gfCNCPoint2[8454] = {X 428.4411, Y 41.5212, Z -3.0000, A 0.000, B 0.000, C 0.000 }
gfCNCPoint2[8455] = {X 429.0371, Y 40.7849, Z -3.0000, A 0.000, B 0.000, C 0.000 }
gfCNCPoint2[8456] = {X 429.7641, Y 40.1776, Z -3.0000, A 0.000, B 0.000, C 0.000 }
gfCNCPoint2[8457] = {X 430.5947, Y 39.7222, Z -3.0000, A 0.000, B 0.000, C 0.000 }
gfCNCPoint2[8458] = {X 434.2534, Y 32.5608, Z -3.0000, A 0.000, B 0.000, C 0.000 }
gfCNCPoint2[8459] = {X 432.9191, Y 31.5580, Z -3.0000, A 0.000, B 0.000, C 0.000 }
gfCNCPoint2[8460] = {X 431.7385, Y 30.3782, Z -3.0000, A 0.000, B 0.000, C 0.000 }
gfCNCPoint2[8461] = {X 430.7348, Y 29.0445, Z -3.0000, A 0.000, B 0.000, C 0.000 }
gfCNCPoint2[8462] = {X 429.9280, Y 27.5834, Z -3.0000, A 0.000, B 0.000, C 0.000 }
gfCNCPoint2[8463] = {X 429.3339, Y 26.0236, Z -3.0000, A 0.000, B 0.000, C 0.000 }
gfCNCPoint2[8464] = {X 428.8998, Y 24.1501, Z -3.0000, A 0.000, B 0.000, C 0.000 }
gfCNCPoint2[8465] = {X 428.6784, Y 22.2397, Z -3.0000, A 0.000, B 0.000, C 0.000 }
gfCNCPoint2[8466] = {X 428.6725, Y 20.3166, Z -3.0000, A 0.000, B 0.000, C 0.000 }
gfCNCPoint2[8467] = {X 428.8821, Y 18.4049, Z -3.0000, A 0.000, B 0.000, C 0.000 }
gfCNCPoint2[8468] = {X 429.3046, Y 16.5287, Z -3.0000, A 0.000, B 0.000, C 0.000 }
gfCNCPoint2[8469] = {X 429.8216, Y 15.0577, Z -3.0000, A 0.000, B 0.000, C 0.000 }
gfCNCPoint2[8470] = {X 430.5198, Y 13.6635, Z -3.0000, A 0.000, B 0.000, C 0.000 }
gfCNCPoint2[8471] = {X 431.3881, Y 12.3684, Z -3.0000, A 0.000, B 0.000, C 0.000 }
gfCNCPoint2[8472] = {X 432.4125, Y 11.1930, Z -3.0000, A 0.000, B 0.000, C 0.000 }
gfCNCPoint2[8473] = {X 433.6947, Y 10.0649, Z -3.0000, A 0.000, B 0.000, C 0.000 }
gfCNCPoint2[8474] = {X 435.1201, Y 9.1243, Z -3.0000, A 0.000, B 0.000, C 0.000 }
gfCNCPoint2[8475] = {X 436.6617, Y 8.3894, Z -3.0000, A 0.000, B 0.000, C 0.000 }
gfCNCPoint2[8476] = {X 438.2899, Y 7.8741, Z -3.0000, A 0.000, B 0.000, C 0.000 }
gfCNCPoint2[8477] = {X 439.9586, Y 7.5566, Z -3.0000, A 0.000, B 0.000, C 0.000 }
gfCNCPoint2[8478] = {X 441.6469, Y 7.3699, Z -3.0000, A 0.000, B 0.000, C 0.000 }
gfCNCPoint2[8479] = {X 443.3446, Y 7.3153, Z -3.0000, A 0.000, B 0.000, C 0.000 }
gfCNCPoint2[8480] = {X 459.4466, Y 7.3112, Z -3.0000, A 0.000, B 0.000, C 0.000 }
gfCNCPoint2[8481] = {X 460.4094, Y 7.4073, Z -3.0000, A 0.000, B 0.000, C 0.000 }
gfCNCPoint2[8482] = {X 461.3341, Y 7.6918, Z -3.0000, A 0.000, B 0.000, C 0.000 }
gfCNCPoint2[8483] = {X 462.1845, Y 8.1534, Z -3.0000, A 0.000, B 0.000, C 0.000 }
gfCNCPoint2[8484] = {X 462.9268, Y 8.7740, Z -3.0000, A 0.000, B 0.000, C 0.000 }
gfCNCPoint2[8485] = {X 463.5318, Y 9.5291, Z -3.0000, A 0.000, B 0.000, C 0.000 }
gfCNCPoint2[8486] = {X 463.9756, Y 10.3888, Z -3.0000, A 0.000, B 0.000, C 0.000 }
gfCNCPoint2[8487] = {X 464.2316, Y 11.2695, Z -3.0000, A 0.000, B 0.000, C 0.000 }
gfCNCPoint2[8488] = {X 464.3179, Y 12.1826, Z -3.0000, A 0.000, B 0.000, C 0.000 }
gfCNCPoint2[8489] = {X 464.3179, Y 12.9779, Z -3.0000, A 0.000, B 0.000, C 0.000 }
gfCNCPoint2[8490] = {X 464.2173, Y 13.9638, Z -3.0000, A 0.000, B 0.000, C 0.000 }
gfCNCPoint2[8491] = {X 463.9196, Y 14.9091, Z -3.0000, A 0.000, B 0.000, C 0.000 }
gfCNCPoint2[8492] = {X 463.4371, Y 15.7747, Z -3.0000, A 0.000, B 0.000, C 0.000 }
gfCNCPoint2[8493] = {X 462.7896, Y 16.5249, Z -3.0000, A 0.000, B 0.000, C 0.000 }
gfCNCPoint2[8494] = {X 462.7893, Y 16.7698, Z -3.0000, A 0.000, B 0.000, C 0.000 }
gfCNCPoint2[8495] = {X 462.7904, Y 40.6626, Z -3.0000, A 0.000, B 0.000, C 0.000 }
gfCNCPoint2[8496] = {X 463.4315, Y 41.4042, Z -3.0000, A 0.000, B 0.000, C 0.000 }
gfCNCPoint2[8497] = {X 463.9115, Y 42.2590, Z -3.0000, A 0.000, B 0.000, C 0.000 }
gfCNCPoint2[8498] = {X 464.2109, Y 43.1925, Z -3.0000, A 0.000, B 0.000, C 0.000 }
gfCNCPoint2[8499] = {X 464.3178, Y 44.1670, Z -3.0000, A 0.000, B 0.000, C 0.000 }
gfCNCPoint2[8500] = {X 464.3179, Y 45.0000, Z -3.0000, A 0.000, B 0.000, C 0.000 }
gfCNCPoint2[8501] = {X 464.3082, Y 45.3090, Z -3.0000, A 0.000, B 0.000, C 0.000 }
gfCNCPoint2[8502] = {X 464.2788, Y 45.6167, Z -3.0000, A 0.000, B 0.000, C 0.000 }
gfCNCPoint2[8503] = {X 464.0485, Y 46.5992, Z -3.0000, A 0.000, B 0.000, C 0.000 }
gfCNCPoint2[8504] = {X 463.6209, Y 47.5134, Z -3.0000, A 0.000, B 0.000, C 0.000 }
gfCNCPoint2[8505] = {X 463.0145, Y 48.3200, Z -3.0000, A 0.000, B 0.000, C 0.000 }
gfCNCPoint2[8506] = {X 462.6627, Y 47.9934, Z -3.0000, A 0.000, B 0.000, C 0.000 }
gfCNCPoint2[8507] = {X 461.9835, Y 48.5889, Z -3.0000, A 0.000, B 0.000, C 0.000 }
gfCNCPoint2[8508] = {X 461.1970, Y 49.0331, Z -3.0000, A 0.000, B 0.000, C 0.000 }
gfCNCPoint2[8509] = {X 460.3364, Y 49.3073, Z -3.0000, A 0.000, B 0.000, C 0.000 }
gfCNCPoint2[8510] = {X 459.4379, Y 49.4000, Z -3.0000, A 0.000, B 0.000, C 0.000 }
gfCNCPoint2[8511] = {X 452.9945, Y 49.4000, Z -3.0000, A 0.000, B 0.000, C 0.000 }
gfCNCPoint2[8512] = {X 452.0154, Y 49.2897, Z -3.0000, A 0.000, B 0.000, C 0.000 }
gfCNCPoint2[8513] = {X 451.0854, Y 48.9643, Z -3.0000, A 0.000, B 0.000, C 0.000 }
gfCNCPoint2[8514] = {X 450.2511, Y 48.4400, Z -3.0000, A 0.000, B 0.000, C 0.000 }
gfCNCPoint2[8515] = {X 449.5544, Y 47.7433, Z -3.0000, A 0.000, B 0.000, C 0.000 }
gfCNCPoint2[8516] = {X 449.0302, Y 46.9091, Z -3.0000, A 0.000, B 0.000, C 0.000 }
gfCNCPoint2[8517] = {X 448.7048, Y 45.9791, Z -3.0000, A 0.000, B 0.000, C 0.000 }
gfCNCPoint2[8518] = {X 448.5945, Y 45.0000, Z -3.0000, A 0.000, B 0.000, C 0.000 }
gfCNCPoint2[8519] = {X 448.5949, Y 44.1483, Z -3.0000, A 0.000, B 0.000, C 0.000 }
gfCNCPoint2[8520] = {X 448.7053, Y 43.2275, Z -3.0000, A 0.000, B 0.000, C 0.000 }
gfCNCPoint2[8521] = {X 449.0063, Y 42.3503, Z -3.0000, A 0.000, B 0.000, C 0.000 }
gfCNCPoint2[8522] = {X 449.4844, Y 41.5556, Z -3.0000, A 0.000, B 0.000, C 0.000 }
gfCNCPoint2[8523] = {X 450.1184, Y 40.8789, Z -3.0000, A 0.000, B 0.000, C 0.000 }
gfCNCPoint2[8524] = {X 450.1184, Y 34.5538, Z -3.0000, A 0.000, B 0.000, C 0.000 }
gfCNCPoint2[8525] = {X 447.5228, Y 34.5538, Z -3.0000, A 0.000, B 0.000, C 0.000 }
gfCNCPoint2[8526] = {X 443.2762, Y 42.8220, Z -3.0000, A 0.000, B 0.000, C 0.000 }
gfCNCPoint2[8527] = {X 443.4440, Y 43.5064, Z -3.0000, A 0.000, B 0.000, C 0.000 }
gfCNCPoint2[8528] = {X 443.5005, Y 44.2089, Z -3.0000, A 0.000, B 0.000, C 0.000 }
gfCNCPoint2[8529] = {X 443.5005, Y 45.0000, Z -3.0000, A 0.000, B 0.000, C 0.000 }
gfCNCPoint2[8530] = {X 443.3902, Y 45.9791, Z -3.0000, A 0.000, B 0.000, C 0.000 }
gfCNCPoint2[8531] = {X 443.0647, Y 46.9091, Z -3.0000, A 0.000, B 0.000, C 0.000 }
gfCNCPoint2[8532] = {X 442.5405, Y 47.7434, Z -3.0000, A 0.000, B 0.000, C 0.000 }
gfCNCPoint2[8533] = {X 441.8438, Y 48.4401, Z -3.0000, A 0.000, B 0.000, C 0.000 }
gfCNCPoint2[8534] = {X 441.0096, Y 48.9643, Z -3.0000, A 0.000, B 0.000, C 0.000 }
gfCNCPoint2[8535] = {X 440.0796, Y 49.2897, Z -3.0000, A 0.000, B 0.000, C 0.000 }
gfCNCPoint2[8536] = {X 439.1005, Y 49.4000, Z -3.0000, A 0.000, B 0.000, C 0.000 }
gfCNCPoint2[8537] = {X 432.5144, Y 49.4000, Z -3.0000, A 0.000, B 0.000, C 0.000 }
gfCNCPoint2[8538] = {X 431.5353, Y 49.2897, Z -3.0000, A 0.000, B 0.000, C 0.000 }
gfCNCPoint2[8539] = {X 430.6053, Y 48.9643, Z -3.0000, A 0.000, B 0.000, C 0.000 }
gfCNCPoint2[8540] = {X 429.7711, Y 48.4401, Z -3.0000, A 0.000, B 0.000, C 0.000 }
gfCNCPoint2[8541] = {X 429.0743, Y 47.7434, Z -3.0000, A 0.000, B 0.000, C 0.000 }
gfCNCPoint2[8542] = {X 428.5501, Y 46.9091, Z -3.0000, A 0.000, B 0.000, C 0.000 }
gfCNCPoint2[8543] = {X 428.2247, Y 45.9791, Z -3.0000, A 0.000, B 0.000, C 0.000 }
gfCNCPoint2[8544] = {X 428.1144, Y 45.0000, Z -3.0000, A 0.000, B 0.000, C 0.000 }
gfCNCPoint2[8545] = {X 428.1148, Y 44.1483, Z -3.0000, A 0.000, B 0.000, C 0.000 }
gfCNCPoint2[8546] = {X 428.2132, Y 43.2816, Z -3.0000, A 0.000, B 0.000, C 0.000 }
gfCNCPoint2[8547] = {X 428.4806, Y 42.4514, Z -3.0000, A 0.000, B 0.000, C 0.000 }
gfCNCPoint2[8548] = {X 428.9065, Y 41.6903, Z -3.0000, A 0.000, B 0.000, C 0.000 }
gfCNCPoint2[8549] = {X 429.4741, Y 41.0281, Z -3.0000, A 0.000, B 0.000, C 0.000 }
gfCNCPoint2[8550] = {X 430.1613, Y 40.4909, Z -3.0000, A 0.000, B 0.000, C 0.000 }
gfCNCPoint2[8551] = {X 430.9408, Y 40.0998, Z -3.0000, A 0.000, B 0.000, C 0.000 }
gfCNCPoint2[8552] = {X 434.8818, Y 32.3858, Z -3.0000, A 0.000, B 0.000, C 0.000 }
gfCNCPoint2[8553] = {X 433.7183, Y 31.5933, Z -3.0000, A 0.000, B 0.000, C 0.000 }
gfCNCPoint2[8554] = {X 432.6614, Y 30.6634, Z -3.0000, A 0.000, B 0.000, C 0.000 }
gfCNCPoint2[8555] = {X 431.7272, Y 29.6103, Z -3.0000, A 0.000, B 0.000, C 0.000 }
gfCNCPoint2[8556] = {X 430.9298, Y 28.4502, Z -3.0000, A 0.000, B 0.000, C 0.000 }
gfCNCPoint2[8557] = {X 430.2815, Y 27.2006, Z -3.0000, A 0.000, B 0.000, C 0.000 }
gfCNCPoint2[8558] = {X 429.7922, Y 25.8807, Z -3.0000, A 0.000, B 0.000, C 0.000 }
gfCNCPoint2[8559] = {X 429.3715, Y 24.0610, Z -3.0000, A 0.000, B 0.000, C 0.000 }
gfCNCPoint2[8560] = {X 429.1572, Y 22.2057, Z -3.0000, A 0.000, B 0.000, C 0.000 }
gfCNCPoint2[8561] = {X 429.1520, Y 20.3381, Z -3.0000, A 0.000, B 0.000, C 0.000 }
gfCNCPoint2[8562] = {X 429.3559, Y 18.4816, Z -3.0000, A 0.000, B 0.000, C 0.000 }
gfCNCPoint2[8563] = {X 429.7664, Y 16.6596, Z -3.0000, A 0.000, B 0.000, C 0.000 }
gfCNCPoint2[8564] = {X 430.2916, Y 15.1794, Z -3.0000, A 0.000, B 0.000, C 0.000 }
gfCNCPoint2[8565] = {X 431.0076, Y 13.7814, Z -3.0000, A 0.000, B 0.000, C 0.000 }
gfCNCPoint2[8566] = {X 431.9019, Y 12.4902, Z -3.0000, A 0.000, B 0.000, C 0.000 }
gfCNCPoint2[8567] = {X 432.9588, Y 11.3283, Z -3.0000, A 0.000, B 0.000, C 0.000 }
gfCNCPoint2[8568] = {X 434.1598, Y 10.3161, Z -3.0000, A 0.000, B 0.000, C 0.000 }
gfCNCPoint2[8569] = {X 435.4839, Y 9.4712, Z -3.0000, A 0.000, B 0.000, C 0.000 }
gfCNCPoint2[8570] = {X 436.9079, Y 8.8085, Z -3.0000, A 0.000, B 0.000, C 0.000 }
gfCNCPoint2[8571] = {X 438.4069, Y 8.3396, Z -3.0000, A 0.000, B 0.000, C 0.000 }
gfCNCPoint2[8572] = {X 440.0370, Y 8.0301, Z -3.0000, A 0.000, B 0.000, C 0.000 }
gfCNCPoint2[8573] = {X 441.6861, Y 7.8483, Z -3.0000, A 0.000, B 0.000, C 0.000 }
gfCNCPoint2[8574] = {X 443.3444, Y 7.7953, Z -3.0000, A 0.000, B 0.000, C 0.000 }
gfCNCPoint2[8575] = {X 444.0367, Y 7.7912, Z -3.0000, A 0.000, B 0.000, C 0.000 }
gfCNCPoint2[8576] = {X 459.4466, Y 7.7912, Z -3.0000, A 0.000, B 0.000, C 0.000 }
gfCNCPoint2[8577] = {X 460.4238, Y 7.9013, Z -3.0000, A 0.000, B 0.000, C 0.000 }
gfCNCPoint2[8578] = {X 461.3519, Y 8.2261, Z -3.0000, A 0.000, B 0.000, C 0.000 }
gfCNCPoint2[8579] = {X 462.1846, Y 8.7493, Z -3.0000, A 0.000, B 0.000, C 0.000 }
gfCNCPoint2[8580] = {X 462.8799, Y 9.4446, Z -3.0000, A 0.000, B 0.000, C 0.000 }
gfCNCPoint2[8581] = {X 463.4031, Y 10.2773, Z -3.0000, A 0.000, B 0.000, C 0.000 }
gfCNCPoint2[8582] = {X 463.7278, Y 11.2054, Z -3.0000, A 0.000, B 0.000, C 0.000 }
gfCNCPoint2[8583] = {X 463.8379, Y 12.1826, Z -3.0000, A 0.000, B 0.000, C 0.000 }
gfCNCPoint2[8584] = {X 463.8377, Y 13.0201, Z -3.0000, A 0.000, B 0.000, C 0.000 }
gfCNCPoint2[8585] = {X 463.7299, Y 13.9472, Z -3.0000, A 0.000, B 0.000, C 0.000 }
gfCNCPoint2[8586] = {X 463.4289, Y 14.8306, Z -3.0000, A 0.000, B 0.000, C 0.000 }
gfCNCPoint2[8587] = {X 462.9484, Y 15.6307, Z -3.0000, A 0.000, B 0.000, C 0.000 }
gfCNCPoint2[8588] = {X 462.3099, Y 16.3115, Z -3.0000, A 0.000, B 0.000, C 0.000 }
gfCNCPoint2[8589] = {X 462.3093, Y 16.7692, Z -3.0000, A 0.000, B 0.000, C 0.000 }
gfCNCPoint2[8590] = {X 462.3104, Y 40.8758, Z -3.0000, A 0.000, B 0.000, C 0.000 }
gfCNCPoint2[8591] = {X 462.9550, Y 41.5649, Z -3.0000, A 0.000, B 0.000, C 0.000 }
gfCNCPoint2[8592] = {X 463.4379, Y 42.3757, Z -3.0000, A 0.000, B 0.000, C 0.000 }
gfCNCPoint2[8593] = {X 463.7368, Y 43.2707, Z -3.0000, A 0.000, B 0.000, C 0.000 }
gfCNCPoint2[8594] = {X 463.8379, Y 44.2089, Z -3.0000, A 0.000, B 0.000, C 0.000 }
gfCNCPoint2[8595] = {X 463.8379, Y 45.0000, Z -3.0000, A 0.000, B 0.000, C 0.000 }
gfCNCPoint2[8596] = {X 463.7612, Y 45.8182, Z -3.0000, A 0.000, B 0.000, C 0.000 }
gfCNCPoint2[8597] = {X 463.5336, Y 46.6079, Z -3.0000, A 0.000, B 0.000, C 0.000 }
gfCNCPoint2[8598] = {X 463.1632, Y 47.3415, Z -3.0000, A 0.000, B 0.000, C 0.000 }
gfCNCPoint2[8599] = {X 462.6627, Y 47.9934, Z -3.0000, A 0.000, B 0.000, C 0.000 }
gfCNCPoint2[8600] = {X 463.0145, Y 48.3200, Z -3.0000, A 0.000, B 0.000, C 0.000 }
gfCNCPoint2[8601] = {X 472.1884, Y 48.3200, Z -3.0000, A 0.000, B 0.000, C 0.000 }
gfCNCPoint2[8602] = {X 471.5820, Y 47.5134, Z -3.0000, A 0.000, B 0.000, C 0.000 }
gfCNCPoint2[8603] = {X 471.1544, Y 46.5992, Z -3.0000, A 0.000, B 0.000, C 0.000 }
gfCNCPoint2[8604] = {X 470.9241, Y 45.6167, Z -3.0000, A 0.000, B 0.000, C 0.000 }
gfCNCPoint2[8605] = {X 470.8947, Y 45.3090, Z -3.0000, A 0.000, B 0.000, C 0.000 }
gfCNCPoint2[8606] = {X 470.8850, Y 45.0000, Z -3.0000, A 0.000, B 0.000, C 0.000 }
gfCNCPoint2[8607] = {X 470.8850, Y 44.2089, Z -3.0000, A 0.000, B 0.000, C 0.000 }
gfCNCPoint2[8608] = {X 470.9769, Y 43.2661, Z -3.0000, A 0.000, B 0.000, C 0.000 }
gfCNCPoint2[8609] = {X 471.2492, Y 42.3588, Z -3.0000, A 0.000, B 0.000, C 0.000 }
gfCNCPoint2[8610] = {X 471.6917, Y 41.5212, Z -3.0000, A 0.000, B 0.000, C 0.000 }
gfCNCPoint2[8611] = {X 472.2877, Y 40.7849, Z -3.0000, A 0.000, B 0.000, C 0.000 }
gfCNCPoint2[8612] = {X 473.0147, Y 40.1776, Z -3.0000, A 0.000, B 0.000, C 0.000 }
gfCNCPoint2[8613] = {X 473.8453, Y 39.7222, Z -3.0000, A 0.000, B 0.000, C 0.000 }
gfCNCPoint2[8614] = {X 477.5004, Y 32.5678, Z -3.0000, A 0.000, B 0.000, C 0.000 }
gfCNCPoint2[8615] = {X 476.2832, Y 31.6578, Z -3.0000, A 0.000, B 0.000, C 0.000 }
gfCNCPoint2[8616] = {X 475.1905, Y 30.6016, Z -3.0000, A 0.000, B 0.000, C 0.000 }
gfCNCPoint2[8617] = {X 474.2397, Y 29.4160, Z -3.0000, A 0.000, B 0.000, C 0.000 }
gfCNCPoint2[8618] = {X 473.4459, Y 28.1201, Z -3.0000, A 0.000, B 0.000, C 0.000 }
gfCNCPoint2[8619] = {X 472.8218, Y 26.7344, Z -3.0000, A 0.000, B 0.000, C 0.000 }
gfCNCPoint2[8620] = {X 472.3774, Y 25.2811, Z -3.0000, A 0.000, B 0.000, C 0.000 }
gfCNCPoint2[8621] = {X 472.0533, Y 23.5418, Z -3.0000, A 0.000, B 0.000, C 0.000 }
gfCNCPoint2[8622] = {X 471.9084, Y 21.7785, Z -3.0000, A 0.000, B 0.000, C 0.000 }
gfCNCPoint2[8623] = {X 471.9443, Y 20.0096, Z -3.0000, A 0.000, B 0.000, C 0.000 }
gfCNCPoint2[8624] = {X 472.1606, Y 18.2537, Z -3.0000, A 0.000, B 0.000, C 0.000 }
gfCNCPoint2[8625] = {X 472.5550, Y 16.5290, Z -3.0000, A 0.000, B 0.000, C 0.000 }
gfCNCPoint2[8626] = {X 473.0735, Y 15.0580, Z -3.0000, A 0.000, B 0.000, C 0.000 }
gfCNCPoint2[8627] = {X 473.7727, Y 13.6638, Z -3.0000, A 0.000, B 0.000, C 0.000 }
gfCNCPoint2[8628] = {X 474.6416, Y 12.3685, Z -3.0000, A 0.000, B 0.000, C 0.000 }
gfCNCPoint2[8629] = {X 475.6663, Y 11.1926, Z -3.0000, A 0.000, B 0.000, C 0.000 }
gfCNCPoint2[8630] = {X 476.7438, Y 10.2237, Z -3.0000, A 0.000, B 0.000, C 0.000 }
gfCNCPoint2[8631] = {X 477.9270, Y 9.3871, Z -3.0000, A 0.000, B 0.000, C 0.000 }
gfCNCPoint2[8632] = {X 479.1998, Y 8.6945, Z -3.0000, A 0.000, B 0.000, C 0.000 }
gfCNCPoint2[8633] = {X 480.5447, Y 8.1552, Z -3.0000, A 0.000, B 0.000, C 0.000 }
gfCNCPoint2[8634] = {X 481.9435, Y 7.7767, Z -3.0000, A 0.000, B 0.000, C 0.000 }
gfCNCPoint2[8635] = {X 484.0947, Y 7.4412, Z -3.0000, A 0.000, B 0.000, C 0.000 }
gfCNCPoint2[8636] = {X 486.2688, Y 7.3234, Z -3.0000, A 0.000, B 0.000, C 0.000 }
gfCNCPoint2[8637] = {X 486.9707, Y 7.3112, Z -3.0000, A 0.000, B 0.000, C 0.000 }
gfCNCPoint2[8638] = {X 502.2122, Y 7.3113, Z -3.0000, A 0.000, B 0.000, C 0.000 }
gfCNCPoint2[8639] = {X 502.7418, Y 7.3154, Z -3.0000, A 0.000, B 0.000, C 0.000 }
gfCNCPoint2[8640] = {X 503.6963, Y 7.4176, Z -3.0000, A 0.000, B 0.000, C 0.000 }
gfCNCPoint2[8641] = {X 504.6121, Y 7.7052, Z -3.0000, A 0.000, B 0.000, C 0.000 }
gfCNCPoint2[8642] = {X 505.4537, Y 8.1670, Z -3.0000, A 0.000, B 0.000, C 0.000 }
gfCNCPoint2[8643] = {X 506.1881, Y 8.7852, Z -3.0000, A 0.000, B 0.000, C 0.000 }
gfCNCPoint2[8644] = {X 506.7869, Y 9.5355, Z -3.0000, A 0.000, B 0.000, C 0.000 }
gfCNCPoint2[8645] = {X 507.2267, Y 10.3887, Z -3.0000, A 0.000, B 0.000, C 0.000 }
gfCNCPoint2[8646] = {X 507.4823, Y 11.2682, Z -3.0000, A 0.000, B 0.000, C 0.000 }
gfCNCPoint2[8647] = {X 507.5685, Y 12.1800, Z -3.0000, A 0.000, B 0.000, C 0.000 }
gfCNCPoint2[8648] = {X 507.5683, Y 13.0237, Z -3.0000, A 0.000, B 0.000, C 0.000 }
gfCNCPoint2[8649] = {X 507.4609, Y 13.9973, Z -3.0000, A 0.000, B 0.000, C 0.000 }
gfCNCPoint2[8650] = {X 507.1612, Y 14.9298, Z -3.0000, A 0.000, B 0.000, C 0.000 }
gfCNCPoint2[8651] = {X 506.6813, Y 15.7837, Z -3.0000, A 0.000, B 0.000, C 0.000 }
gfCNCPoint2[8652] = {X 506.0406, Y 16.5245, Z -3.0000, A 0.000, B 0.000, C 0.000 }
gfCNCPoint2[8653] = {X 506.0405, Y 40.6622, Z -3.0000, A 0.000, B 0.000, C 0.000 }
gfCNCPoint2[8654] = {X 506.6818, Y 41.4038, Z -3.0000, A 0.000, B 0.000, C 0.000 }
gfCNCPoint2[8655] = {X 507.1618, Y 42.2585, Z -3.0000, A 0.000, B 0.000, C 0.000 }
gfCNCPoint2[8656] = {X 507.4614, Y 43.1920, Z -3.0000, A 0.000, B 0.000, C 0.000 }
gfCNCPoint2[8657] = {X 507.5683, Y 44.1665, Z -3.0000, A 0.000, B 0.000, C 0.000 }
gfCNCPoint2[8658] = {X 507.5685, Y 45.0000, Z -3.0000, A 0.000, B 0.000, C 0.000 }
gfCNCPoint2[8659] = {X 507.4747, Y 45.9520, Z -3.0000, A 0.000, B 0.000, C 0.000 }
gfCNCPoint2[8660] = {X 507.1970, Y 46.8675, Z -3.0000, A 0.000, B 0.000, C 0.000 }
gfCNCPoint2[8661] = {X 506.7461, Y 47.7112, Z -3.0000, A 0.000, B 0.000, C 0.000 }
gfCNCPoint2[8662] = {X 506.1392, Y 48.4507, Z -3.0000, A 0.000, B 0.000, C 0.000 }
gfCNCPoint2[8663] = {X 505.3997, Y 49.0576, Z -3.0000, A 0.000, B 0.000, C 0.000 }
gfCNCPoint2[8664] = {X 504.5560, Y 49.5085, Z -3.0000, A 0.000, B 0.000, C 0.000 }
gfCNCPoint2[8665] = {X 503.6405, Y 49.7862, Z -3.0000, A 0.000, B 0.000, C 0.000 }
gfCNCPoint2[8666] = {X 502.6885, Y 49.8800, Z -3.0000, A 0.000, B 0.000, C 0.000 }
gfCNCPoint2[8667] = {X 496.2450, Y 49.8800, Z -3.0000, A 0.000, B 0.000, C 0.000 }
gfCNCPoint2[8668] = {X 495.2220, Y 49.7716, Z -3.0000, A 0.000, B 0.000, C 0.000 }
gfCNCPoint2[8669] = {X 494.2445, Y 49.4511, Z -3.0000, A 0.000, B 0.000, C 0.000 }
gfCNCPoint2[8670] = {X 493.3559, Y 48.9328, Z -3.0000, A 0.000, B 0.000, C 0.000 }
gfCNCPoint2[8671] = {X 492.5956, Y 48.2398, Z -3.0000, A 0.000, B 0.000, C 0.000 }
gfCNCPoint2[8672] = {X 491.9976, Y 47.4028, Z -3.0000, A 0.000, B 0.000, C 0.000 }
gfCNCPoint2[8673] = {X 491.5882, Y 46.4590, Z -3.0000, A 0.000, B 0.000, C 0.000 }
gfCNCPoint2[8674] = {X 491.4241, Y 45.7570, Z -3.0000, A 0.000, B 0.000, C 0.000 }
gfCNCPoint2[8675] = {X 491.3652, Y 45.0385, Z -3.0000, A 0.000, B 0.000, C 0.000 }
gfCNCPoint2[8676] = {X 491.3655, Y 44.1416, Z -3.0000, A 0.000, B 0.000, C 0.000 }
gfCNCPoint2[8677] = {X 491.4758, Y 43.1751, Z -3.0000, A 0.000, B 0.000, C 0.000 }
gfCNCPoint2[8678] = {X 491.7756, Y 42.2496, Z -3.0000, A 0.000, B 0.000, C 0.000 }
gfCNCPoint2[8679] = {X 492.2530, Y 41.4020, Z -3.0000, A 0.000, B 0.000, C 0.000 }
gfCNCPoint2[8680] = {X 492.8890, Y 40.6660, Z -3.0000, A 0.000, B 0.000, C 0.000 }
gfCNCPoint2[8681] = {X 492.8890, Y 35.0338, Z -3.0000, A 0.000, B 0.000, C 0.000 }
gfCNCPoint2[8682] = {X 491.0658, Y 35.0338, Z -3.0000, A 0.000, B 0.000, C 0.000 }
gfCNCPoint2[8683] = {X 487.0430, Y 42.8673, Z -3.0000, A 0.000, B 0.000, C 0.000 }
gfCNCPoint2[8684] = {X 487.1807, Y 43.5098, Z -3.0000, A 0.000, B 0.000, C 0.000 }
gfCNCPoint2[8685] = {X 487.2308, Y 44.1648, Z -3.0000, A 0.000, B 0.000, C 0.000 }
gfCNCPoint2[8686] = {X 487.2310, Y 45.0000, Z -3.0000, A 0.000, B 0.000, C 0.000 }
gfCNCPoint2[8687] = {X 487.1749, Y 45.7380, Z -3.0000, A 0.000, B 0.000, C 0.000 }
gfCNCPoint2[8688] = {X 487.0078, Y 46.4590, Z -3.0000, A 0.000, B 0.000, C 0.000 }
gfCNCPoint2[8689] = {X 486.5939, Y 47.4110, Z -3.0000, A 0.000, B 0.000, C 0.000 }
gfCNCPoint2[8690] = {X 485.9879, Y 48.2538, Z -3.0000, A 0.000, B 0.000, C 0.000 }
gfCNCPoint2[8691] = {X 485.2175, Y 48.9494, Z -3.0000, A 0.000, B 0.000, C 0.000 }
gfCNCPoint2[8692] = {X 484.3173, Y 49.4663, Z -3.0000, A 0.000, B 0.000, C 0.000 }
gfCNCPoint2[8693] = {X 483.3557, Y 49.7755, Z -3.0000, A 0.000, B 0.000, C 0.000 }
gfCNCPoint2[8694] = {X 482.3510, Y 49.8800, Z -3.0000, A 0.000, B 0.000, C 0.000 }
gfCNCPoint2[8695] = {X 480.2695, Y 49.8800, Z -3.0000, A 0.000, B 0.000, C 0.000 }
gfCNCPoint2[8696] = {X 480.2695, Y 49.4000, Z -3.0000, A 0.000, B 0.000, C 0.000 }
gfCNCPoint2[8697] = {X 475.7650, Y 49.4000, Z -3.0000, A 0.000, B 0.000, C 0.000 }
gfCNCPoint2[8698] = {X 474.7859, Y 49.2897, Z -3.0000, A 0.000, B 0.000, C 0.000 }
gfCNCPoint2[8699] = {X 473.8559, Y 48.9643, Z -3.0000, A 0.000, B 0.000, C 0.000 }
gfCNCPoint2[8700] = {X 473.0216, Y 48.4401, Z -3.0000, A 0.000, B 0.000, C 0.000 }
gfCNCPoint2[8701] = {X 472.3249, Y 47.7434, Z -3.0000, A 0.000, B 0.000, C 0.000 }
gfCNCPoint2[8702] = {X 471.8007, Y 46.9091, Z -3.0000, A 0.000, B 0.000, C 0.000 }
gfCNCPoint2[8703] = {X 471.4753, Y 45.9791, Z -3.0000, A 0.000, B 0.000, C 0.000 }
gfCNCPoint2[8704] = {X 471.3650, Y 45.0000, Z -3.0000, A 0.000, B 0.000, C 0.000 }
gfCNCPoint2[8705] = {X 471.3654, Y 44.1483, Z -3.0000, A 0.000, B 0.000, C 0.000 }
gfCNCPoint2[8706] = {X 471.4638, Y 43.2816, Z -3.0000, A 0.000, B 0.000, C 0.000 }
gfCNCPoint2[8707] = {X 471.7311, Y 42.4514, Z -3.0000, A 0.000, B 0.000, C 0.000 }
gfCNCPoint2[8708] = {X 472.1570, Y 41.6903, Z -3.0000, A 0.000, B 0.000, C 0.000 }
gfCNCPoint2[8709] = {X 472.7247, Y 41.0281, Z -3.0000, A 0.000, B 0.000, C 0.000 }
gfCNCPoint2[8710] = {X 473.4118, Y 40.4909, Z -3.0000, A 0.000, B 0.000, C 0.000 }
gfCNCPoint2[8711] = {X 474.1914, Y 40.0998, Z -3.0000, A 0.000, B 0.000, C 0.000 }
gfCNCPoint2[8712] = {X 478.1278, Y 32.3948, Z -3.0000, A 0.000, B 0.000, C 0.000 }
gfCNCPoint2[8713] = {X 476.8711, Y 31.5206, Z -3.0000, A 0.000, B 0.000, C 0.000 }
gfCNCPoint2[8714] = {X 475.7412, Y 30.4878, Z -3.0000, A 0.000, B 0.000, C 0.000 }
gfCNCPoint2[8715] = {X 474.7577, Y 29.3148, Z -3.0000, A 0.000, B 0.000, C 0.000 }
gfCNCPoint2[8716] = {X 473.9379, Y 28.0219, Z -3.0000, A 0.000, B 0.000, C 0.000 }
gfCNCPoint2[8717] = {X 473.2964, Y 26.6320, Z -3.0000, A 0.000, B 0.000, C 0.000 }
gfCNCPoint2[8718] = {X 472.8443, Y 25.1695, Z -3.0000, A 0.000, B 0.000, C 0.000 }
gfCNCPoint2[8719] = {X 472.5291, Y 23.4784, Z -3.0000, A 0.000, B 0.000, C 0.000 }
gfCNCPoint2[8720] = {X 472.3882, Y 21.7639, Z -3.0000, A 0.000, B 0.000, C 0.000 }
gfCNCPoint2[8721] = {X 472.4231, Y 20.0440, Z -3.0000, A 0.000, B 0.000, C 0.000 }
gfCNCPoint2[8722] = {X 472.6334, Y 18.3367, Z -3.0000, A 0.000, B 0.000, C 0.000 }
gfCNCPoint2[8723] = {X 473.0168, Y 16.6598, Z -3.0000, A 0.000, B 0.000, C 0.000 }
gfCNCPoint2[8724] = {X 473.5631, Y 15.1347, Z -3.0000, A 0.000, B 0.000, C 0.000 }
gfCNCPoint2[8725] = {X 474.3113, Y 13.6979, Z -3.0000, A 0.000, B 0.000, C 0.000 }
gfCNCPoint2[8726] = {X 475.2476, Y 12.3759, Z -3.0000, A 0.000, B 0.000, C 0.000 }
gfCNCPoint2[8727] = {X 476.3546, Y 11.1932, Z -3.0000, A 0.000, B 0.000, C 0.000 }
gfCNCPoint2[8728] = {X 477.6119, Y 10.1717, Z -3.0000, A 0.000, B 0.000, C 0.000 }
gfCNCPoint2[8729] = {X 478.9963, Y 9.3304, Z -3.0000, A 0.000, B 0.000, C 0.000 }
gfCNCPoint2[8730] = {X 480.4820, Y 8.6847, Z -3.0000, A 0.000, B 0.000, C 0.000 }
gfCNCPoint2[8731] = {X 482.0416, Y 8.2466, Z -3.0000, A 0.000, B 0.000, C 0.000 }
gfCNCPoint2[8732] = {X 484.1466, Y 7.9184, Z -3.0000, A 0.000, B 0.000, C 0.000 }
gfCNCPoint2[8733] = {X 486.2739, Y 7.8034, Z -3.0000, A 0.000, B 0.000, C 0.000 }
gfCNCPoint2[8734] = {X 486.9707, Y 7.7912, Z -3.0000, A 0.000, B 0.000, C 0.000 }
gfCNCPoint2[8735] = {X 502.2084, Y 7.7912, Z -3.0000, A 0.000, B 0.000, C 0.000 }
gfCNCPoint2[8736] = {X 502.7380, Y 7.7954, Z -3.0000, A 0.000, B 0.000, C 0.000 }
gfCNCPoint2[8737] = {X 503.7081, Y 7.9118, Z -3.0000, A 0.000, B 0.000, C 0.000 }
gfCNCPoint2[8738] = {X 504.6282, Y 8.2401, Z -3.0000, A 0.000, B 0.000, C 0.000 }
gfCNCPoint2[8739] = {X 505.4529, Y 8.7641, Z -3.0000, A 0.000, B 0.000, C 0.000 }
gfCNCPoint2[8740] = {X 506.1410, Y 9.4576, Z -3.0000, A 0.000, B 0.000, C 0.000 }
gfCNCPoint2[8741] = {X 506.6585, Y 10.2863, Z -3.0000, A 0.000, B 0.000, C 0.000 }
gfCNCPoint2[8742] = {X 506.9796, Y 11.2091, Z -3.0000, A 0.000, B 0.000, C 0.000 }
gfCNCPoint2[8743] = {X 507.0885, Y 12.1800, Z -3.0000, A 0.000, B 0.000, C 0.000 }
gfCNCPoint2[8744] = {X 507.0883, Y 13.0233, Z -3.0000, A 0.000, B 0.000, C 0.000 }
gfCNCPoint2[8745] = {X 506.9799, Y 13.9495, Z -3.0000, A 0.000, B 0.000, C 0.000 }
gfCNCPoint2[8746] = {X 506.6788, Y 14.8320, Z -3.0000, A 0.000, B 0.000, C 0.000 }
gfCNCPoint2[8747] = {X 506.1985, Y 15.6312, Z -3.0000, A 0.000, B 0.000, C 0.000 }
gfCNCPoint2[8748] = {X 505.5606, Y 16.3113, Z -3.0000, A 0.000, B 0.000, C 0.000 }
gfCNCPoint2[8749] = {X 505.5605, Y 40.8754, Z -3.0000, A 0.000, B 0.000, C 0.000 }
gfCNCPoint2[8750] = {X 506.2053, Y 41.5646, Z -3.0000, A 0.000, B 0.000, C 0.000 }
gfCNCPoint2[8751] = {X 506.6883, Y 42.3754, Z -3.0000, A 0.000, B 0.000, C 0.000 }
gfCNCPoint2[8752] = {X 506.9873, Y 43.2706, Z -3.0000, A 0.000, B 0.000, C 0.000 }
gfCNCPoint2[8753] = {X 507.0885, Y 44.2089, Z -3.0000, A 0.000, B 0.000, C 0.000 }
gfCNCPoint2[8754] = {X 507.0885, Y 45.0000, Z -3.0000, A 0.000, B 0.000, C 0.000 }
gfCNCPoint2[8755] = {X 506.9782, Y 45.9791, Z -3.0000, A 0.000, B 0.000, C 0.000 }
gfCNCPoint2[8756] = {X 506.6528, Y 46.9091, Z -3.0000, A 0.000, B 0.000, C 0.000 }
gfCNCPoint2[8757] = {X 506.1285, Y 47.7434, Z -3.0000, A 0.000, B 0.000, C 0.000 }
gfCNCPoint2[8758] = {X 505.4318, Y 48.4401, Z -3.0000, A 0.000, B 0.000, C 0.000 }
gfCNCPoint2[8759] = {X 504.5976, Y 48.9643, Z -3.0000, A 0.000, B 0.000, C 0.000 }
gfCNCPoint2[8760] = {X 503.6676, Y 49.2897, Z -3.0000, A 0.000, B 0.000, C 0.000 }
gfCNCPoint2[8761] = {X 502.6885, Y 49.4000, Z -3.0000, A 0.000, B 0.000, C 0.000 }
gfCNCPoint2[8762] = {X 496.2450, Y 49.4000, Z -3.0000, A 0.000, B 0.000, C 0.000 }
gfCNCPoint2[8763] = {X 495.2659, Y 49.2897, Z -3.0000, A 0.000, B 0.000, C 0.000 }
gfCNCPoint2[8764] = {X 494.3359, Y 48.9643, Z -3.0000, A 0.000, B 0.000, C 0.000 }
gfCNCPoint2[8765] = {X 493.5017, Y 48.4400, Z -3.0000, A 0.000, B 0.000, C 0.000 }
gfCNCPoint2[8766] = {X 492.8050, Y 47.7433, Z -3.0000, A 0.000, B 0.000, C 0.000 }
gfCNCPoint2[8767] = {X 492.2807, Y 46.9091, Z -3.0000, A 0.000, B 0.000, C 0.000 }
gfCNCPoint2[8768] = {X 491.9553, Y 45.9791, Z -3.0000, A 0.000, B 0.000, C 0.000 }
gfCNCPoint2[8769] = {X 491.8450, Y 45.0000, Z -3.0000, A 0.000, B 0.000, C 0.000 }
gfCNCPoint2[8770] = {X 491.8454, Y 44.1483, Z -3.0000, A 0.000, B 0.000, C 0.000 }
gfCNCPoint2[8771] = {X 491.9559, Y 43.2275, Z -3.0000, A 0.000, B 0.000, C 0.000 }
gfCNCPoint2[8772] = {X 492.2568, Y 42.3503, Z -3.0000, A 0.000, B 0.000, C 0.000 }
gfCNCPoint2[8773] = {X 492.7349, Y 41.5556, Z -3.0000, A 0.000, B 0.000, C 0.000 }
gfCNCPoint2[8774] = {X 493.3690, Y 40.8789, Z -3.0000, A 0.000, B 0.000, C 0.000 }
gfCNCPoint2[8775] = {X 493.3690, Y 34.5538, Z -3.0000, A 0.000, B 0.000, C 0.000 }
gfCNCPoint2[8776] = {X 490.7727, Y 34.5538, Z -3.0000, A 0.000, B 0.000, C 0.000 }
gfCNCPoint2[8777] = {X 486.5267, Y 42.8219, Z -3.0000, A 0.000, B 0.000, C 0.000 }
gfCNCPoint2[8778] = {X 486.6946, Y 43.5064, Z -3.0000, A 0.000, B 0.000, C 0.000 }
gfCNCPoint2[8779] = {X 486.7510, Y 44.2089, Z -3.0000, A 0.000, B 0.000, C 0.000 }
gfCNCPoint2[8780] = {X 486.7510, Y 45.0000, Z -3.0000, A 0.000, B 0.000, C 0.000 }
gfCNCPoint2[8781] = {X 486.6407, Y 45.9791, Z -3.0000, A 0.000, B 0.000, C 0.000 }
gfCNCPoint2[8782] = {X 486.3153, Y 46.9091, Z -3.0000, A 0.000, B 0.000, C 0.000 }
gfCNCPoint2[8783] = {X 485.7911, Y 47.7434, Z -3.0000, A 0.000, B 0.000, C 0.000 }
gfCNCPoint2[8784] = {X 485.0944, Y 48.4401, Z -3.0000, A 0.000, B 0.000, C 0.000 }
gfCNCPoint2[8785] = {X 484.2601, Y 48.9643, Z -3.0000, A 0.000, B 0.000, C 0.000 }
gfCNCPoint2[8786] = {X 483.3301, Y 49.2897, Z -3.0000, A 0.000, B 0.000, C 0.000 }
gfCNCPoint2[8787] = {X 482.3510, Y 49.4000, Z -3.0000, A 0.000, B 0.000, C 0.000 }
gfCNCPoint2[8788] = {X 480.2695, Y 49.4000, Z -3.0000, A 0.000, B 0.000, C 0.000 }
gfCNCPoint2[8789] = {X 480.2695, Y 49.8800, Z -3.0000, A 0.000, B 0.000, C 0.000 }
gfCNCPoint2[8790] = {X 481.4067, Y 50.7435, Z -3.0000, A 0.000, B 0.000, C 0.000 }
gfCNCPoint2[8791] = {X 482.4044, Y 51.7649, Z -3.0000, A 0.000, B 0.000, C 0.000 }
gfCNCPoint2[8792] = {X 483.2411, Y 52.9219, Z -3.0000, A 0.000, B 0.000, C 0.000 }
gfCNCPoint2[8793] = {X 483.8615, Y 54.1044, Z -3.0000, A 0.000, B 0.000, C 0.000 }
gfCNCPoint2[8794] = {X 484.3133, Y 55.3610, Z -3.0000, A 0.000, B 0.000, C 0.000 }
gfCNCPoint2[8795] = {X 484.5879, Y 56.6678, Z -3.0000, A 0.000, B 0.000, C 0.000 }
gfCNCPoint2[8796] = {X 484.6800, Y 58.0000, Z -3.0000, A 0.000, B 0.000, C 0.000 }
gfCNCPoint2[8797] = {X 484.6797, Y 59.0140, Z -3.0000, A 0.000, B 0.000, C 0.000 }
gfCNCPoint2[8798] = {X 484.5592, Y 60.4585, Z -3.0000, A 0.000, B 0.000, C 0.000 }
gfCNCPoint2[8799] = {X 484.2244, Y 61.8688, Z -3.0000, A 0.000, B 0.000, C 0.000 }
gfCNCPoint2[8800] = {X 483.6828, Y 63.2133, Z -3.0000, A 0.000, B 0.000, C 0.000 }
gfCNCPoint2[8801] = {X 482.9464, Y 64.4618, Z -3.0000, A 0.000, B 0.000, C 0.000 }
gfCNCPoint2[8802] = {X 482.0319, Y 65.5864, Z -3.0000, A 0.000, B 0.000, C 0.000 }
gfCNCPoint2[8803] = {X 480.9598, Y 66.5619, Z -3.0000, A 0.000, B 0.000, C 0.000 }
gfCNCPoint2[8804] = {X 480.9601, Y 89.4448, Z -3.0000, A 0.000, B 0.000, C 0.000 }
gfCNCPoint2[8805] = {X 482.0597, Y 90.4470, Z -3.0000, A 0.000, B 0.000, C 0.000 }
gfCNCPoint2[8806] = {X 482.9922, Y 91.6062, Z -3.0000, A 0.000, B 0.000, C 0.000 }
gfCNCPoint2[8807] = {X 483.7355, Y 92.8950, Z -3.0000, A 0.000, B 0.000, C 0.000 }
gfCNCPoint2[8808] = {X 507.6818, Y 92.8950, Z -3.0000, A 0.000, B 0.000, C 0.000 }
gfCNCPoint2[8809] = {X 507.6818, Y 95.2950, Z -3.0000, A 0.000, B 0.000, C 0.000 }
gfCNCPoint2[8810] = {X 595.2965, Y 95.2950, Z -3.0000, A 0.000, B 0.000, C 0.000 }
gfCNCPoint2[8811] = {X 595.2965, Y 54.2000, Z -3.0000, A 0.000, B 0.000, C 0.000 }
gfCNCPoint2[8812] = {X 593.5565, Y 54.2000, Z -3.0000, A 0.000, B 0.000, C 0.000 }
gfCNCPoint2[8813] = {X 592.2403, Y 54.1053, Z -3.0000, A 0.000, B 0.000, C 0.000 }
gfCNCPoint2[8814] = {X 590.9511, Y 53.8233, Z -3.0000, A 0.000, B 0.000, C 0.000 }
gfCNCPoint2[8815] = {X 589.7155, Y 53.3598, Z -3.0000, A 0.000, B 0.000, C 0.000 }
gfCNCPoint2[8816] = {X 588.5589, Y 52.7242, Z -3.0000, A 0.000, B 0.000, C 0.000 }
gfCNCPoint2[8817] = {X 587.5052, Y 51.9297, Z -3.0000, A 0.000, B 0.000, C 0.000 }
gfCNCPoint2[8818] = {X 586.4956, Y 52.6955, Z -3.0000, A 0.000, B 0.000, C 0.000 }
gfCNCPoint2[8819] = {X 585.3903, Y 53.3153, Z -3.0000, A 0.000, B 0.000, C 0.000 }
gfCNCPoint2[8820] = {X 584.1375, Y 53.7999, Z -3.0000, A 0.000, B 0.000, C 0.000 }
gfCNCPoint2[8821] = {X 582.8276, Y 54.0969, Z -3.0000, A 0.000, B 0.000, C 0.000 }
gfCNCPoint2[8822] = {X 581.4884, Y 54.1999, Z -3.0000, A 0.000, B 0.000, C 0.000 }
gfCNCPoint2[8823] = {X 580.1485, Y 54.1069, Z -3.0000, A 0.000, B 0.000, C 0.000 }
gfCNCPoint2[8824] = {X 578.8364, Y 53.8198, Z -3.0000, A 0.000, B 0.000, C 0.000 }
gfCNCPoint2[8825] = {X 577.5801, Y 53.3447, Z -3.0000, A 0.000, B 0.000, C 0.000 }
gfCNCPoint2[8826] = {X 576.4063, Y 52.6917, Z -3.0000, A 0.000, B 0.000, C 0.000 }
gfCNCPoint2[8827] = {X 575.3401, Y 51.8748, Z -3.0000, A 0.000, B 0.000, C 0.000 }
gfCNCPoint2[8828] = {X 574.2798, Y 52.6879, Z -3.0000, A 0.000, B 0.000, C 0.000 }
gfCNCPoint2[8829] = {X 573.1128, Y 53.3388, Z -3.0000, A 0.000, B 0.000, C 0.000 }
gfCNCPoint2[8830] = {X 571.8638, Y 53.8139, Z -3.0000, A 0.000, B 0.000, C 0.000 }
gfCNCPoint2[8831] = {X 570.5592, Y 54.1030, Z -3.0000, A 0.000, B 0.000, C 0.000 }
gfCNCPoint2[8832] = {X 569.2264, Y 54.2000, Z -3.0000, A 0.000, B 0.000, C 0.000 }
gfCNCPoint2[8833] = {X 562.4443, Y 54.2000, Z -3.0000, A 0.000, B 0.000, C 0.000 }
gfCNCPoint2[8834] = {X 561.0051, Y 54.0867, Z -3.0000, A 0.000, B 0.000, C 0.000 }
gfCNCPoint2[8835] = {X 559.6013, Y 53.7497, Z -3.0000, A 0.000, B 0.000, C 0.000 }
gfCNCPoint2[8836] = {X 558.2676, Y 53.1973, Z -3.0000, A 0.000, B 0.000, C 0.000 }
gfCNCPoint2[8837] = {X 557.0367, Y 52.4430, Z -3.0000, A 0.000, B 0.000, C 0.000 }
gfCNCPoint2[8838] = {X 555.9389, Y 51.5054, Z -3.0000, A 0.000, B 0.000, C 0.000 }
gfCNCPoint2[8839] = {X 555.0013, Y 50.4076, Z -3.0000, A 0.000, B 0.000, C 0.000 }
gfCNCPoint2[8840] = {X 554.2470, Y 49.1767, Z -3.0000, A 0.000, B 0.000, C 0.000 }
gfCNCPoint2[8841] = {X 553.6946, Y 47.8430, Z -3.0000, A 0.000, B 0.000, C 0.000 }
gfCNCPoint2[8842] = {X 553.3576, Y 46.4392, Z -3.0000, A 0.000, B 0.000, C 0.000 }
gfCNCPoint2[8843] = {X 553.2443, Y 45.0000, Z -3.0000, A 0.000, B 0.000, C 0.000 }
gfCNCPoint2[8844] = {X 553.2443, Y 44.0599, Z -3.0000, A 0.000, B 0.000, C 0.000 }
gfCNCPoint2[8845] = {X 553.3451, Y 42.7237, Z -3.0000, A 0.000, B 0.000, C 0.000 }
gfCNCPoint2[8846] = {X 553.6381, Y 41.4162, Z -3.0000, A 0.000, B 0.000, C 0.000 }
gfCNCPoint2[8847] = {X 554.1172, Y 40.1649, Z -3.0000, A 0.000, B 0.000, C 0.000 }
gfCNCPoint2[8848] = {X 554.7724, Y 38.9960, Z -3.0000, A 0.000, B 0.000, C 0.000 }
gfCNCPoint2[8849] = {X 554.7724, Y 11.0116, Z -3.0000, A 0.000, B 0.000, C 0.000 }
gfCNCPoint2[8850] = {X 554.1221, Y 9.8560, Z -3.0000, A 0.000, B 0.000, C 0.000 }
gfCNCPoint2[8851] = {X 553.6448, Y 8.6189, Z -3.0000, A 0.000, B 0.000, C 0.000 }
gfCNCPoint2[8852] = {X 553.3502, Y 7.3261, Z -3.0000, A 0.000, B 0.000, C 0.000 }
gfCNCPoint2[8853] = {X 553.2446, Y 6.0043, Z -3.0000, A 0.000, B 0.000, C 0.000 }
gfCNCPoint2[8854] = {X 553.2443, Y 5.0000, Z -3.0000, A 0.000, B 0.000, C 0.000 }
gfCNCPoint2[8855] = {X 553.2455, Y 4.8525, Z -3.0000, A 0.000, B 0.000, C 0.000 }
gfCNCPoint2[8856] = {X 553.2490, Y 4.7050, Z -3.0000, A 0.000, B 0.000, C 0.000 }
gfCNCPoint2[8857] = {X 365.1865, Y 4.7050, Z -3.0000, A 0.000, B 0.000, C 0.000 }
gfCNCPoint2[8858] = {X 365.5704, Y 5.1228, Z -3.0000, A 0.000, B 0.000, C 0.000 }
gfCNCPoint2[8859] = {X 365.9444, Y 5.5496, Z -3.0000, A 0.000, B 0.000, C 0.000 }
gfCNCPoint2[8860] = {X 367.0648, Y 6.9483, Z -3.0000, A 0.000, B 0.000, C 0.000 }
gfCNCPoint2[8861] = {X 368.0923, Y 8.4167, Z -3.0000, A 0.000, B 0.000, C 0.000 }
gfCNCPoint2[8862] = {X 369.3424, Y 10.5319, Z -3.0000, A 0.000, B 0.000, C 0.000 }
gfCNCPoint2[8863] = {X 370.4001, Y 12.7498, Z -3.0000, A 0.000, B 0.000, C 0.000 }
gfCNCPoint2[8864] = {X 371.2569, Y 15.0526, Z -3.0000, A 0.000, B 0.000, C 0.000 }
gfCNCPoint2[8865] = {X 371.9061, Y 17.4224, Z -3.0000, A 0.000, B 0.000, C 0.000 }
gfCNCPoint2[8866] = {X 372.3615, Y 19.8203, Z -3.0000, A 0.000, B 0.000, C 0.000 }
gfCNCPoint2[8867] = {X 372.6467, Y 22.2444, Z -3.0000, A 0.000, B 0.000, C 0.000 }
gfCNCPoint2[8868] = {X 372.7601, Y 24.6825, Z -3.0000, A 0.000, B 0.000, C 0.000 }
gfCNCPoint2[8869] = {X 372.7014, Y 27.1226, Z -3.0000, A 0.000, B 0.000, C 0.000 }
gfCNCPoint2[8870] = {X 372.4707, Y 29.5525, Z -3.0000, A 0.000, B 0.000, C 0.000 }
gfCNCPoint2[8871] = {X 372.0692, Y 31.9600, Z -3.0000, A 0.000, B 0.000, C 0.000 }
gfCNCPoint2[8872] = {X 371.4823, Y 34.3171, Z -3.0000, A 0.000, B 0.000, C 0.000 }
gfCNCPoint2[8873] = {X 370.6896, Y 36.6131, Z -3.0000, A 0.000, B 0.000, C 0.000 }
gfCNCPoint2[8874] = {X 369.6973, Y 38.8302, Z -3.0000, A 0.000, B 0.000, C 0.000 }
gfCNCPoint2[8875] = {X 368.5130, Y 40.9509, Z -3.0000, A 0.000, B 0.000, C 0.000 }
gfCNCPoint2[8876] = {X 367.1460, Y 42.9588, Z -3.0000, A 0.000, B 0.000, C 0.000 }
gfCNCPoint2[8877] = {X 365.7530, Y 44.6742, Z -3.0000, A 0.000, B 0.000, C 0.000 }
gfCNCPoint2[8878] = {X 364.2148, Y 46.2607, Z -3.0000, A 0.000, B 0.000, C 0.000 }
gfCNCPoint2[8879] = {X 362.5433, Y 47.7060, Z -3.0000, A 0.000, B 0.000, C 0.000 }
gfCNCPoint2[8880] = {X 360.7513, Y 48.9989, Z -3.0000, A 0.000, B 0.000, C 0.000 }
gfCNCPoint2[8881] = {X 358.8527, Y 50.1296, Z -3.0000, A 0.000, B 0.000, C 0.000 }
gfCNCPoint2[8882] = {X 356.6377, Y 51.1398, Z -3.0000, A 0.000, B 0.000, C 0.000 }
gfCNCPoint2[8883] = {X 354.3368, Y 51.9349, Z -3.0000, A 0.000, B 0.000, C 0.000 }
gfCNCPoint2[8884] = {X 351.9708, Y 52.5078, Z -3.0000, A 0.000, B 0.000, C 0.000 }
gfCNCPoint2[8885] = {X 349.5610, Y 52.8533, Z -3.0000, A 0.000, B 0.000, C 0.000 }
gfCNCPoint2[8886] = {X 347.1293, Y 52.9683, Z -3.0000, A 0.000, B 0.000, C 0.000 }
gfCNCPoint2[8887] = {X 344.8097, Y 52.9257, Z -3.0000, A 0.000, B 0.000, C 0.000 }
gfCNCPoint2[8888] = {X 342.5025, Y 52.6824, Z -3.0000, A 0.000, B 0.000, C 0.000 }
gfCNCPoint2[8889] = {X 340.2251, Y 52.2402, Z -3.0000, A 0.000, B 0.000, C 0.000 }
gfCNCPoint2[8890] = {X 337.9945, Y 51.6025, Z -3.0000, A 0.000, B 0.000, C 0.000 }
gfCNCPoint2[8891] = {X 335.8275, Y 50.7740, Z -3.0000, A 0.000, B 0.000, C 0.000 }
gfCNCPoint2[8892] = {X 333.7404, Y 49.7610, Z -3.0000, A 0.000, B 0.000, C 0.000 }
gfCNCPoint2[8893] = {X 332.8334, Y 49.2270, Z -3.0000, A 0.000, B 0.000, C 0.000 }
gfCNCPoint2[8894] = {X 331.9481, Y 48.6579, Z -3.0000, A 0.000, B 0.000, C 0.000 }
gfCNCPoint2[8895] = {X 331.3028, Y 48.2111, Z -3.0000, A 0.000, B 0.000, C 0.000 }
gfCNCPoint2[8896] = {X 330.6709, Y 47.7456, Z -3.0000, A 0.000, B 0.000, C 0.000 }
gfCNCPoint2[8897] = {X 329.2194, Y 49.6569, Z -3.0000, A 0.000, B 0.000, C 0.000 }
gfCNCPoint2[8898] = {X 328.8738, Y 49.3903, Z -3.0000, A 0.000, B 0.000, C 0.000 }
gfCNCPoint2[8899] = {X 328.5322, Y 49.1187, Z -3.0000, A 0.000, B 0.000, C 0.000 }
gfCNCPoint2[8900] = {X 328.1269, Y 49.0391, Z -3.0000, A 0.000, B 0.000, C 0.000 }
gfCNCPoint2[8901] = {X 327.7253, Y 48.9423, Z -3.0000, A 0.000, B 0.000, C 0.000 }
gfCNCPoint2[8902] = {X 328.4876, Y 49.2676, Z -3.0000, A 0.000, B 0.000, C 0.000 }
gfCNCPoint2[8903] = {X 329.2194, Y 49.6569, Z -3.0000, A 0.000, B 0.000, C 0.000 }
gfCNCPoint2[8904] = {X 330.6709, Y 47.7456, Z -3.0000, A 0.000, B 0.000, C 0.000 }
gfCNCPoint2[8905] = {X 330.0963, Y 47.2968, Z -3.0000, A 0.000, B 0.000, C 0.000 }
gfCNCPoint2[8906] = {X 329.5341, Y 46.8324, Z -3.0000, A 0.000, B 0.000, C 0.000 }
gfCNCPoint2[8907] = {X 328.9313, Y 46.7520, Z -3.0000, A 0.000, B 0.000, C 0.000 }
gfCNCPoint2[8908] = {X 328.3374, Y 46.6216, Z -3.0000, A 0.000, B 0.000, C 0.000 }
gfCNCPoint2[8909] = {X 327.9789, Y 46.5172, Z -3.0000, A 0.000, B 0.000, C 0.000 }
gfCNCPoint2[8910] = {X 327.6263, Y 46.3944, Z -3.0000, A 0.000, B 0.000, C 0.000 }
gfCNCPoint2[8911] = {X 326.7320, Y 45.9864, Z -3.0000, A 0.000, B 0.000, C 0.000 }
gfCNCPoint2[8912] = {X 325.9009, Y 45.4616, Z -3.0000, A 0.000, B 0.000, C 0.000 }
gfCNCPoint2[8913] = {X 325.1480, Y 44.8296, Z -3.0000, A 0.000, B 0.000, C 0.000 }
gfCNCPoint2[8914] = {X 324.5140, Y 44.2115, Z -3.0000, A 0.000, B 0.000, C 0.000 }
gfCNCPoint2[8915] = {X 324.0475, Y 43.7117, Z -3.0000, A 0.000, B 0.000, C 0.000 }
gfCNCPoint2[8916] = {X 323.6300, Y 43.1703, Z -3.0000, A 0.000, B 0.000, C 0.000 }
gfCNCPoint2[8917] = {X 319.6957, Y 45.9200, Z -3.0000, A 0.000, B 0.000, C 0.000 }
gfCNCPoint2[8918] = {X 319.4780, Y 45.5976, Z -3.0000, A 0.000, B 0.000, C 0.000 }
gfCNCPoint2[8919] = {X 319.2708, Y 45.2683, Z -3.0000, A 0.000, B 0.000, C 0.000 }
gfCNCPoint2[8920] = {X 319.2514, Y 45.5948, Z -3.0000, A 0.000, B 0.000, C 0.000 }
gfCNCPoint2[8921] = {X 319.2174, Y 45.9200, Z -3.0000, A 0.000, B 0.000, C 0.000 }
gfCNCPoint2[8922] = {X 319.6957, Y 45.9200, Z -3.0000, A 0.000, B 0.000, C 0.000 }
gfCNCPoint2[8923] = {X 321.6628, Y 44.5452, Z -3.0000, A 0.000, B 0.000, C 0.000 }
gfCNCPoint2[8924] = {X 321.4884, Y 44.2868, Z -3.0000, A 0.000, B 0.000, C 0.000 }
gfCNCPoint2[8925] = {X 321.3224, Y 44.0230, Z -3.0000, A 0.000, B 0.000, C 0.000 }
gfCNCPoint2[8926] = {X 320.6713, Y 42.7458, Z -3.0000, A 0.000, B 0.000, C 0.000 }
gfCNCPoint2[8927] = {X 320.2159, Y 41.3864, Z -3.0000, A 0.000, B 0.000, C 0.000 }
gfCNCPoint2[8928] = {X 319.9664, Y 39.9747, Z -3.0000, A 0.000, B 0.000, C 0.000 }
gfCNCPoint2[8929] = {X 319.9280, Y 38.5416, Z -3.0000, A 0.000, B 0.000, C 0.000 }
gfCNCPoint2[8930] = {X 320.1018, Y 37.1186, Z -3.0000, A 0.000, B 0.000, C 0.000 }
gfCNCPoint2[8931] = {X 320.4298, Y 35.8917, Z -3.0000, A 0.000, B 0.000, C 0.000 }
gfCNCPoint2[8932] = {X 320.9156, Y 34.7183, Z -3.0000, A 0.000, B 0.000, C 0.000 }
gfCNCPoint2[8933] = {X 321.5508, Y 33.6186, Z -3.0000, A 0.000, B 0.000, C 0.000 }
gfCNCPoint2[8934] = {X 324.1375, Y 29.7509, Z -3.0000, A 0.000, B 0.000, C 0.000 }
gfCNCPoint2[8935] = {X 320.1476, Y 27.0825, Z -3.0000, A 0.000, B 0.000, C 0.000 }
gfCNCPoint2[8936] = {X 321.7941, Y 24.6207, Z -3.0000, A 0.000, B 0.000, C 0.000 }
gfCNCPoint2[8937] = {X 321.9845, Y 24.3429, Z -3.0000, A 0.000, B 0.000, C 0.000 }
gfCNCPoint2[8938] = {X 322.1814, Y 24.0697, Z -3.0000, A 0.000, B 0.000, C 0.000 }
gfCNCPoint2[8939] = {X 321.5380, Y 23.0773, Z -3.0000, A 0.000, B 0.000, C 0.000 }
gfCNCPoint2[8940] = {X 320.9778, Y 22.0356, Z -3.0000, A 0.000, B 0.000, C 0.000 }
gfCNCPoint2[8941] = {X 320.1477, Y 20.3280, Z -3.0000, A 0.000, B 0.000, C 0.000 }
gfCNCPoint2[8942] = {X 320.1476, Y 27.0825, Z -3.0000, A 0.000, B 0.000, C 0.000 }
gfCNCPoint2[8943] = {X 322.1426, Y 28.4167, Z -3.0000, A 0.000, B 0.000, C 0.000 }
gfCNCPoint2[8944] = {X 323.7890, Y 25.9549, Z -3.0000, A 0.000, B 0.000, C 0.000 }
gfCNCPoint2[8945] = {X 324.5064, Y 24.9899, Z -3.0000, A 0.000, B 0.000, C 0.000 }
gfCNCPoint2[8946] = {X 325.3162, Y 24.1010, Z -3.0000, A 0.000, B 0.000, C 0.000 }
gfCNCPoint2[8947] = {X 324.4812, Y 23.1413, Z -3.0000, A 0.000, B 0.000, C 0.000 }
gfCNCPoint2[8948] = {X 323.7518, Y 22.0990, Z -3.0000, A 0.000, B 0.000, C 0.000 }
gfCNCPoint2[8949] = {X 323.1360, Y 20.9859, Z -3.0000, A 0.000, B 0.000, C 0.000 }
gfCNCPoint2[8950] = {X 319.6151, Y 13.7428, Z -3.0000, A 0.000, B 0.000, C 0.000 }
gfCNCPoint2[8951] = {X 319.4387, Y 13.3633, Z -3.0000, A 0.000, B 0.000, C 0.000 }
gfCNCPoint2[8952] = {X 319.2755, Y 12.9779, Z -3.0000, A 0.000, B 0.000, C 0.000 }
gfCNCPoint2[8953] = {X 319.2755, Y 13.0353, Z -3.0000, A 0.000, B 0.000, C 0.000 }
gfCNCPoint2[8954] = {X 319.1697, Y 14.2158, Z -3.0000, A 0.000, B 0.000, C 0.000 }
gfCNCPoint2[8955] = {X 318.8738, Y 15.3634, Z -3.0000, A 0.000, B 0.000, C 0.000 }
gfCNCPoint2[8956] = {X 318.3956, Y 16.4479, Z -3.0000, A 0.000, B 0.000, C 0.000 }
gfCNCPoint2[8957] = {X 317.7477, Y 17.4404, Z -3.0000, A 0.000, B 0.000, C 0.000 }
gfCNCPoint2[8958] = {X 317.7475, Y 36.6521, Z -3.0000, A 0.000, B 0.000, C 0.000 }
gfCNCPoint2[8959] = {X 318.1569, Y 35.1211, Z -3.0000, A 0.000, B 0.000, C 0.000 }
gfCNCPoint2[8960] = {X 318.7631, Y 33.6568, Z -3.0000, A 0.000, B 0.000, C 0.000 }
gfCNCPoint2[8961] = {X 319.5559, Y 32.2844, Z -3.0000, A 0.000, B 0.000, C 0.000 }
gfCNCPoint2[8962] = {X 322.1426, Y 28.4167, Z -3.0000, A 0.000, B 0.000, C 0.000 }
gfCNCPoint2[8963] = {X 324.1375, Y 29.7509, Z -3.0000, A 0.000, B 0.000, C 0.000 }
gfCNCPoint2[8964] = {X 325.7840, Y 27.2891, Z -3.0000, A 0.000, B 0.000, C 0.000 }
gfCNCPoint2[8965] = {X 326.3588, Y 26.5158, Z -3.0000, A 0.000, B 0.000, C 0.000 }
gfCNCPoint2[8966] = {X 327.0077, Y 25.8035, Z -3.0000, A 0.000, B 0.000, C 0.000 }
gfCNCPoint2[8967] = {X 328.0707, Y 24.8904, Z -3.0000, A 0.000, B 0.000, C 0.000 }
gfCNCPoint2[8968] = {X 329.2543, Y 24.1403, Z -3.0000, A 0.000, B 0.000, C 0.000 }
gfCNCPoint2[8969] = {X 328.0859, Y 23.3667, Z -3.0000, A 0.000, B 0.000, C 0.000 }
gfCNCPoint2[8970] = {X 327.0414, Y 22.4326, Z -3.0000, A 0.000, B 0.000, C 0.000 }
gfCNCPoint2[8971] = {X 326.3723, Y 21.6635, Z -3.0000, A 0.000, B 0.000, C 0.000 }
gfCNCPoint2[8972] = {X 325.7878, Y 20.8284, Z -3.0000, A 0.000, B 0.000, C 0.000 }
gfCNCPoint2[8973] = {X 325.2944, Y 19.9364, Z -3.0000, A 0.000, B 0.000, C 0.000 }
gfCNCPoint2[8974] = {X 321.7736, Y 12.6936, Z -3.0000, A 0.000, B 0.000, C 0.000 }
gfCNCPoint2[8975] = {X 321.6322, Y 12.3894, Z -3.0000, A 0.000, B 0.000, C 0.000 }
gfCNCPoint2[8976] = {X 321.5015, Y 12.0806, Z -3.0000, A 0.000, B 0.000, C 0.000 }
gfCNCPoint2[8977] = {X 321.1058, Y 10.8774, Z -3.0000, A 0.000, B 0.000, C 0.000 }
gfCNCPoint2[8978] = {X 320.8706, Y 9.6328, Z -3.0000, A 0.000, B 0.000, C 0.000 }
gfCNCPoint2[8979] = {X 320.7999, Y 8.3681, Z -3.0000, A 0.000, B 0.000, C 0.000 }
gfCNCPoint2[8980] = {X 320.8950, Y 7.1050, Z -3.0000, A 0.000, B 0.000, C 0.000 }
gfCNCPoint2[8981] = {X 298.7842, Y 7.1050, Z -3.0000, A 0.000, B 0.000, C 0.000 }
gfCNCPoint2[8982] = {X 298.7842, Y 9.5050, Z -3.0000, A 0.000, B 0.000, C 0.000 }
gfCNCPoint2[8983] = {X 297.8292, Y 9.5050, Z -3.0000, A 0.000, B 0.000, C 0.000 }
gfCNCPoint2[8984] = {X 298.1371, Y 10.4755, Z -3.0000, A 0.000, B 0.000, C 0.000 }
gfCNCPoint2[8985] = {X 298.3067, Y 11.4795, Z -3.0000, A 0.000, B 0.000, C 0.000 }
gfCNCPoint2[8986] = {X 298.4762, Y 10.4755, Z -3.0000, A 0.000, B 0.000, C 0.000 }
gfCNCPoint2[8987] = {X 298.7842, Y 9.5050, Z -3.0000, A 0.000, B 0.000, C 0.000 }
gfCNCPoint2[8988] = {X 298.7842, Y 7.1050, Z -3.0000, A 0.000, B 0.000, C 0.000 }
gfCNCPoint2[8989] = {X 233.3050, Y 7.1050, Z -3.0000, A 0.000, B 0.000, C 0.000 }
gfCNCPoint2[8990] = {X 233.3050, Y 11.9050, Z -3.0000, A 0.000, B 0.000, C 0.000 }
gfCNCPoint2[8991] = {X 233.1564, Y 11.9050, Z -3.0000, A 0.000, B 0.000, C 0.000 }
gfCNCPoint2[8992] = {X 233.1594, Y 12.0455, Z -3.0000, A 0.000, B 0.000, C 0.000 }
gfCNCPoint2[8993] = {X 233.1605, Y 12.1859, Z -3.0000, A 0.000, B 0.000, C 0.000 }
gfCNCPoint2[8994] = {X 233.2321, Y 12.0452, Z -3.0000, A 0.000, B 0.000, C 0.000 }
gfCNCPoint2[8995] = {X 233.3050, Y 11.9050, Z -3.0000, A 0.000, B 0.000, C 0.000 }
gfCNCPoint2[8996] = {X 233.3050, Y 9.5050, Z -3.0000, A 0.000, B 0.000, C 0.000 }
gfCNCPoint2[8997] = {X 230.2485, Y 9.5050, Z -3.0000, A 0.000, B 0.000, C 0.000 }
gfCNCPoint2[8998] = {X 230.6107, Y 10.7178, Z -3.0000, A 0.000, B 0.000, C 0.000 }
gfCNCPoint2[8999] = {X 230.7574, Y 11.9749, Z -3.0000, A 0.000, B 0.000, C 0.000 }
gfCNCPoint2[9000] = {X 230.7597, Y 12.0808, Z -3.0000, A 0.000, B 0.000, C 0.000 }
gfCNCPoint2[9001] = {X 230.7605, Y 12.1868, Z -3.0000, A 0.000, B 0.000, C 0.000 }
gfCNCPoint2[9002] = {X 230.7602, Y 13.0462, Z -3.0000, A 0.000, B 0.000, C 0.000 }
gfCNCPoint2[9003] = {X 230.6531, Y 14.2237, Z -3.0000, A 0.000, B 0.000, C 0.000 }
gfCNCPoint2[9004] = {X 230.3568, Y 15.3684, Z -3.0000, A 0.000, B 0.000, C 0.000 }
gfCNCPoint2[9005] = {X 229.8792, Y 16.4501, Z -3.0000, A 0.000, B 0.000, C 0.000 }
gfCNCPoint2[9006] = {X 229.2327, Y 17.4401, Z -3.0000, A 0.000, B 0.000, C 0.000 }
gfCNCPoint2[9007] = {X 229.2330, Y 25.8453, Z -3.0000, A 0.000, B 0.000, C 0.000 }
gfCNCPoint2[9008] = {X 231.6330, Y 25.8452, Z -3.0000, A 0.000, B 0.000, C 0.000 }
gfCNCPoint2[9009] = {X 231.6335, Y 38.9904, Z -3.0000, A 0.000, B 0.000, C 0.000 }
gfCNCPoint2[9010] = {X 231.6440, Y 39.0069, Z -3.0000, A 0.000, B 0.000, C 0.000 }
gfCNCPoint2[9011] = {X 232.3931, Y 37.9855, Z -3.0000, A 0.000, B 0.000, C 0.000 }
gfCNCPoint2[9012] = {X 233.2692, Y 37.0706, Z -3.0000, A 0.000, B 0.000, C 0.000 }
gfCNCPoint2[9013] = {X 234.2573, Y 36.2780, Z -3.0000, A 0.000, B 0.000, C 0.000 }
gfCNCPoint2[9014] = {X 235.5695, Y 33.7094, Z -3.0000, A 0.000, B 0.000, C 0.000 }
gfCNCPoint2[9015] = {X 234.4289, Y 32.2853, Z -3.0000, A 0.000, B 0.000, C 0.000 }
gfCNCPoint2[9016] = {X 233.4506, Y 30.7450, Z -3.0000, A 0.000, B 0.000, C 0.000 }
gfCNCPoint2[9017] = {X 232.6465, Y 29.1071, Z -3.0000, A 0.000, B 0.000, C 0.000 }
gfCNCPoint2[9018] = {X 232.0261, Y 27.3911, Z -3.0000, A 0.000, B 0.000, C 0.000 }
gfCNCPoint2[9019] = {X 231.8155, Y 26.6217, Z -3.0000, A 0.000, B 0.000, C 0.000 }
gfCNCPoint2[9020] = {X 231.6330, Y 25.8452, Z -3.0000, A 0.000, B 0.000, C 0.000 }
gfCNCPoint2[9021] = {X 229.2330, Y 25.8453, Z -3.0000, A 0.000, B 0.000, C 0.000 }
gfCNCPoint2[9022] = {X 229.2335, Y 39.7477, Z -3.0000, A 0.000, B 0.000, C 0.000 }
gfCNCPoint2[9023] = {X 229.4331, Y 40.0177, Z -3.0000, A 0.000, B 0.000, C 0.000 }
gfCNCPoint2[9024] = {X 229.6200, Y 40.2966, Z -3.0000, A 0.000, B 0.000, C 0.000 }
gfCNCPoint2[9025] = {X 230.1055, Y 41.1910, Z -3.0000, A 0.000, B 0.000, C 0.000 }
gfCNCPoint2[9026] = {X 230.4616, Y 42.1443, Z -3.0000, A 0.000, B 0.000, C 0.000 }
gfCNCPoint2[9027] = {X 230.6813, Y 43.1379, Z -3.0000, A 0.000, B 0.000, C 0.000 }
gfCNCPoint2[9028] = {X 230.7603, Y 44.1524, Z -3.0000, A 0.000, B 0.000, C 0.000 }
gfCNCPoint2[9029] = {X 230.7605, Y 45.0000, Z -3.0000, A 0.000, B 0.000, C 0.000 }
gfCNCPoint2[9030] = {X 230.7459, Y 45.4609, Z -3.0000, A 0.000, B 0.000, C 0.000 }
gfCNCPoint2[9031] = {X 230.7021, Y 45.9200, Z -3.0000, A 0.000, B 0.000, C 0.000 }
gfCNCPoint2[9032] = {X 232.5859, Y 45.9200, Z -3.0000, A 0.000, B 0.000, C 0.000 }
gfCNCPoint2[9033] = {X 232.5421, Y 45.4609, Z -3.0000, A 0.000, B 0.000, C 0.000 }
gfCNCPoint2[9034] = {X 232.5275, Y 45.0000, Z -3.0000, A 0.000, B 0.000, C 0.000 }
gfCNCPoint2[9035] = {X 232.5275, Y 44.2090, Z -3.0000, A 0.000, B 0.000, C 0.000 }
gfCNCPoint2[9036] = {X 232.6006, Y 43.1798, Z -3.0000, A 0.000, B 0.000, C 0.000 }
gfCNCPoint2[9037] = {X 232.8184, Y 42.1714, Z -3.0000, A 0.000, B 0.000, C 0.000 }
gfCNCPoint2[9038] = {X 233.1766, Y 41.2038, Z -3.0000, A 0.000, B 0.000, C 0.000 }
gfCNCPoint2[9039] = {X 233.6680, Y 40.2966, Z -3.0000, A 0.000, B 0.000, C 0.000 }
gfCNCPoint2[9040] = {X 234.3527, Y 39.3876, Z -3.0000, A 0.000, B 0.000, C 0.000 }
gfCNCPoint2[9041] = {X 235.1707, Y 38.5964, Z -3.0000, A 0.000, B 0.000, C 0.000 }
gfCNCPoint2[9042] = {X 236.1021, Y 37.9424, Z -3.0000, A 0.000, B 0.000, C 0.000 }
gfCNCPoint2[9043] = {X 238.5001, Y 33.2484, Z -3.0000, A 0.000, B 0.000, C 0.000 }
gfCNCPoint2[9044] = {X 237.3864, Y 32.1407, Z -3.0000, A 0.000, B 0.000, C 0.000 }
gfCNCPoint2[9045] = {X 236.4012, Y 30.9173, Z -3.0000, A 0.000, B 0.000, C 0.000 }
gfCNCPoint2[9046] = {X 235.5563, Y 29.5931, Z -3.0000, A 0.000, B 0.000, C 0.000 }
gfCNCPoint2[9047] = {X 234.8620, Y 28.1841, Z -3.0000, A 0.000, B 0.000, C 0.000 }
gfCNCPoint2[9048] = {X 234.3267, Y 26.7074, Z -3.0000, A 0.000, B 0.000, C 0.000 }
gfCNCPoint2[9049] = {X 234.1404, Y 26.0262, Z -3.0000, A 0.000, B 0.000, C 0.000 }
gfCNCPoint2[9050] = {X 233.9790, Y 25.3388, Z -3.0000, A 0.000, B 0.000, C 0.000 }
gfCNCPoint2[9051] = {X 233.6675, Y 23.4512, Z -3.0000, A 0.000, B 0.000, C 0.000 }
gfCNCPoint2[9052] = {X 233.5427, Y 21.5421, Z -3.0000, A 0.000, B 0.000, C 0.000 }
gfCNCPoint2[9053] = {X 233.6055, Y 19.6300, Z -3.0000, A 0.000, B 0.000, C 0.000 }
gfCNCPoint2[9054] = {X 233.8554, Y 17.7332, Z -3.0000, A 0.000, B 0.000, C 0.000 }
gfCNCPoint2[9055] = {X 234.2901, Y 15.8701, Z -3.0000, A 0.000, B 0.000, C 0.000 }
gfCNCPoint2[9056] = {X 234.7357, Y 14.5431, Z -3.0000, A 0.000, B 0.000, C 0.000 }
gfCNCPoint2[9057] = {X 235.3047, Y 13.2640, Z -3.0000, A 0.000, B 0.000, C 0.000 }
gfCNCPoint2[9058] = {X 235.3663, Y 13.1429, Z -3.0000, A 0.000, B 0.000, C 0.000 }
gfCNCPoint2[9059] = {X 235.4290, Y 13.0223, Z -3.0000, A 0.000, B 0.000, C 0.000 }
gfCNCPoint2[9060] = {X 236.1704, Y 11.7671, Z -3.0000, A 0.000, B 0.000, C 0.000 }
gfCNCPoint2[9061] = {X 237.0315, Y 10.5909, Z -3.0000, A 0.000, B 0.000, C 0.000 }
gfCNCPoint2[9062] = {X 238.0041, Y 9.5050, Z -3.0000, A 0.000, B 0.000, C 0.000 }
gfCNCPoint2[9063] = {X 233.3050, Y 9.5050, Z -3.0000, A 0.000, B 0.000, C 0.000 }
gfCNCPoint2[9064] = {X 233.3050, Y 7.1050, Z -3.0000, A 0.000, B 0.000, C 0.000 }
gfCNCPoint2[9065] = {X 207.3611, Y 7.1050, Z -3.0000, A 0.000, B 0.000, C 0.000 }
gfCNCPoint2[9066] = {X 207.3611, Y 11.9050, Z -3.0000, A 0.000, B 0.000, C 0.000 }
gfCNCPoint2[9067] = {X 205.8556, Y 11.9050, Z -3.0000, A 0.000, B 0.000, C 0.000 }
gfCNCPoint2[9068] = {X 206.6106, Y 13.3410, Z -3.0000, A 0.000, B 0.000, C 0.000 }
gfCNCPoint2[9069] = {X 207.2363, Y 14.8379, Z -3.0000, A 0.000, B 0.000, C 0.000 }
gfCNCPoint2[9070] = {X 207.7974, Y 16.7110, Z -3.0000, A 0.000, B 0.000, C 0.000 }
gfCNCPoint2[9071] = {X 208.1764, Y 18.6291, Z -3.0000, A 0.000, B 0.000, C 0.000 }
gfCNCPoint2[9072] = {X 208.3698, Y 20.5748, Z -3.0000, A 0.000, B 0.000, C 0.000 }
gfCNCPoint2[9073] = {X 208.3760, Y 22.5300, Z -3.0000, A 0.000, B 0.000, C 0.000 }
gfCNCPoint2[9074] = {X 208.1948, Y 24.4769, Z -3.0000, A 0.000, B 0.000, C 0.000 }
gfCNCPoint2[9075] = {X 207.8279, Y 26.3974, Z -3.0000, A 0.000, B 0.000, C 0.000 }
gfCNCPoint2[9076] = {X 207.3609, Y 28.0096, Z -3.0000, A 0.000, B 0.000, C 0.000 }
gfCNCPoint2[9077] = {X 206.7377, Y 29.5682, Z -3.0000, A 0.000, B 0.000, C 0.000 }
gfCNCPoint2[9078] = {X 205.9642, Y 31.0579, Z -3.0000, A 0.000, B 0.000, C 0.000 }
gfCNCPoint2[9079] = {X 206.0463, Y 31.2162, Z -3.0000, A 0.000, B 0.000, C 0.000 }
gfCNCPoint2[9080] = {X 206.1255, Y 31.3761, Z -3.0000, A 0.000, B 0.000, C 0.000 }
gfCNCPoint2[9081] = {X 208.8855, Y 37.0782, Z -3.0000, A 0.000, B 0.000, C 0.000 }
gfCNCPoint2[9082] = {X 208.8855, Y 18.1987, Z -3.0000, A 0.000, B 0.000, C 0.000 }
gfCNCPoint2[9083] = {X 208.2333, Y 17.0025, Z -3.0000, A 0.000, B 0.000, C 0.000 }
gfCNCPoint2[9084] = {X 207.7554, Y 15.7266, Z -3.0000, A 0.000, B 0.000, C 0.000 }
gfCNCPoint2[9085] = {X 207.4615, Y 14.3962, Z -3.0000, A 0.000, B 0.000, C 0.000 }
gfCNCPoint2[9086] = {X 207.3572, Y 13.0378, Z -3.0000, A 0.000, B 0.000, C 0.000 }
gfCNCPoint2[9087] = {X 207.3570, Y 12.1868, Z -3.0000, A 0.000, B 0.000, C 0.000 }
gfCNCPoint2[9088] = {X 207.3580, Y 12.0459, Z -3.0000, A 0.000, B 0.000, C 0.000 }
gfCNCPoint2[9089] = {X 207.3611, Y 11.9050, Z -3.0000, A 0.000, B 0.000, C 0.000 }
gfCNCPoint2[9090] = {X 207.3611, Y 9.5050, Z -3.0000, A 0.000, B 0.000, C 0.000 }
gfCNCPoint2[9091] = {X 200.9066, Y 9.5050, Z -3.0000, A 0.000, B 0.000, C 0.000 }
gfCNCPoint2[9092] = {X 201.9800, Y 10.6137, Z -3.0000, A 0.000, B 0.000, C 0.000 }
gfCNCPoint2[9093] = {X 202.9416, Y 11.8206, Z -3.0000, A 0.000, B 0.000, C 0.000 }
gfCNCPoint2[9094] = {X 203.7826, Y 13.1145, Z -3.0000, A 0.000, B 0.000, C 0.000 }
gfCNCPoint2[9095] = {X 204.4360, Y 14.3564, Z -3.0000, A 0.000, B 0.000, C 0.000 }
gfCNCPoint2[9096] = {X 204.9781, Y 15.6507, Z -3.0000, A 0.000, B 0.000, C 0.000 }
gfCNCPoint2[9097] = {X 205.5507, Y 17.6374, Z -3.0000, A 0.000, B 0.000, C 0.000 }
gfCNCPoint2[9098] = {X 205.8915, Y 19.6767, Z -3.0000, A 0.000, B 0.000, C 0.000 }
gfCNCPoint2[9099] = {X 205.9960, Y 21.7416, Z -3.0000, A 0.000, B 0.000, C 0.000 }
gfCNCPoint2[9100] = {X 205.8628, Y 23.8049, Z -3.0000, A 0.000, B 0.000, C 0.000 }
gfCNCPoint2[9101] = {X 205.4937, Y 25.8392, Z -3.0000, A 0.000, B 0.000, C 0.000 }
gfCNCPoint2[9102] = {X 205.0926, Y 27.2254, Z -3.0000, A 0.000, B 0.000, C 0.000 }
gfCNCPoint2[9103] = {X 204.5572, Y 28.5654, Z -3.0000, A 0.000, B 0.000, C 0.000 }
gfCNCPoint2[9104] = {X 203.8925, Y 29.8462, Z -3.0000, A 0.000, B 0.000, C 0.000 }
gfCNCPoint2[9105] = {X 203.1051, Y 31.0555, Z -3.0000, A 0.000, B 0.000, C 0.000 }
gfCNCPoint2[9106] = {X 203.5732, Y 31.7147, Z -3.0000, A 0.000, B 0.000, C 0.000 }
gfCNCPoint2[9107] = {X 203.9653, Y 32.4217, Z -3.0000, A 0.000, B 0.000, C 0.000 }
gfCNCPoint2[9108] = {X 206.9865, Y 38.6634, Z -3.0000, A 0.000, B 0.000, C 0.000 }
gfCNCPoint2[9109] = {X 207.4240, Y 39.8017, Z -3.0000, A 0.000, B 0.000, C 0.000 }
gfCNCPoint2[9110] = {X 207.6653, Y 40.9971, Z -3.0000, A 0.000, B 0.000, C 0.000 }
gfCNCPoint2[9111] = {X 207.7038, Y 42.2159, Z -3.0000, A 0.000, B 0.000, C 0.000 }
gfCNCPoint2[9112] = {X 207.5382, Y 43.4241, Z -3.0000, A 0.000, B 0.000, C 0.000 }
gfCNCPoint2[9113] = {X 207.1733, Y 44.5877, Z -3.0000, A 0.000, B 0.000, C 0.000 }
gfCNCPoint2[9114] = {X 206.6193, Y 45.6741, Z -3.0000, A 0.000, B 0.000, C 0.000 }
gfCNCPoint2[9115] = {X 205.8917, Y 46.6527, Z -3.0000, A 0.000, B 0.000, C 0.000 }
gfCNCPoint2[9116] = {X 205.0110, Y 47.4962, Z -3.0000, A 0.000, B 0.000, C 0.000 }
gfCNCPoint2[9117] = {X 204.4733, Y 47.9309, Z -3.0000, A 0.000, B 0.000, C 0.000 }
gfCNCPoint2[9118] = {X 203.5890, Y 48.5430, Z -3.0000, A 0.000, B 0.000, C 0.000 }
gfCNCPoint2[9119] = {X 202.6244, Y 49.0184, Z -3.0000, A 0.000, B 0.000, C 0.000 }
gfCNCPoint2[9120] = {X 201.4897, Y 49.3726, Z -3.0000, A 0.000, B 0.000, C 0.000 }
gfCNCPoint2[9121] = {X 200.3127, Y 49.5378, Z -3.0000, A 0.000, B 0.000, C 0.000 }
gfCNCPoint2[9122] = {X 199.1244, Y 49.5097, Z -3.0000, A 0.000, B 0.000, C 0.000 }
gfCNCPoint2[9123] = {X 196.8334, Y 50.6064, Z -3.0000, A 0.000, B 0.000, C 0.000 }
gfCNCPoint2[9124] = {X 194.4618, Y 51.5159, Z -3.0000, A 0.000, B 0.000, C 0.000 }
gfCNCPoint2[9125] = {X 192.0250, Y 52.2324, Z -3.0000, A 0.000, B 0.000, C 0.000 }
gfCNCPoint2[9126] = {X 190.7220, Y 52.5180, Z -3.0000, A 0.000, B 0.000, C 0.000 }
gfCNCPoint2[9127] = {X 189.4059, Y 52.7353, Z -3.0000, A 0.000, B 0.000, C 0.000 }
gfCNCPoint2[9128] = {X 189.9004, Y 53.9110, Z -3.0000, A 0.000, B 0.000, C 0.000 }
gfCNCPoint2[9129] = {X 190.2682, Y 55.1323, Z -3.0000, A 0.000, B 0.000, C 0.000 }
gfCNCPoint2[9130] = {X 190.5269, Y 56.5558, Z -3.0000, A 0.000, B 0.000, C 0.000 }
gfCNCPoint2[9131] = {X 190.6135, Y 58.0000, Z -3.0000, A 0.000, B 0.000, C 0.000 }
gfCNCPoint2[9132] = {X 190.6132, Y 58.8771, Z -3.0000, A 0.000, B 0.000, C 0.000 }
gfCNCPoint2[9133] = {X 208.6248, Y 78.5344, Z -3.0000, A 0.000, B 0.000, C 0.000 }
gfCNCPoint2[9134] = {X 212.1638, Y 75.2916, Z -3.0000, A 0.000, B 0.000, C 0.000 }
gfCNCPoint2[9135] = {X 215.1994, Y 78.6046, Z -3.0000, A 0.000, B 0.000, C 0.000 }
gfCNCPoint2[9136] = {X 218.3286, Y 76.5998, Z -3.0000, A 0.000, B 0.000, C 0.000 }
gfCNCPoint2[9137] = {X 216.9971, Y 76.0773, Z -3.0000, A 0.000, B 0.000, C 0.000 }
gfCNCPoint2[9138] = {X 216.3768, Y 75.8848, Z -3.0000, A 0.000, B 0.000, C 0.000 }
gfCNCPoint2[9139] = {X 215.7326, Y 75.8035, Z -3.0000, A 0.000, B 0.000, C 0.000 }
gfCNCPoint2[9140] = {X 213.9345, Y 75.6431, Z -3.0000, A 0.000, B 0.000, C 0.000 }
gfCNCPoint2[9141] = {X 212.1638, Y 75.2916, Z -3.0000, A 0.000, B 0.000, C 0.000 }
gfCNCPoint2[9142] = {X 210.3943, Y 76.9130, Z -3.0000, A 0.000, B 0.000, C 0.000 }
gfCNCPoint2[9143] = {X 214.7939, Y 81.7146, Z -3.0000, A 0.000, B 0.000, C 0.000 }
gfCNCPoint2[9144] = {X 223.5832, Y 76.0838, Z -3.0000, A 0.000, B 0.000, C 0.000 }
gfCNCPoint2[9145] = {X 217.8861, Y 73.8479, Z -3.0000, A 0.000, B 0.000, C 0.000 }
gfCNCPoint2[9146] = {X 216.8724, Y 73.5365, Z -3.0000, A 0.000, B 0.000, C 0.000 }
gfCNCPoint2[9147] = {X 215.8202, Y 73.4051, Z -3.0000, A 0.000, B 0.000, C 0.000 }
gfCNCPoint2[9148] = {X 214.2765, Y 73.2676, Z -3.0000, A 0.000, B 0.000, C 0.000 }
gfCNCPoint2[9149] = {X 212.7562, Y 72.9659, Z -3.0000, A 0.000, B 0.000, C 0.000 }
gfCNCPoint2[9150] = {X 211.1572, Y 72.4583, Z -3.0000, A 0.000, B 0.000, C 0.000 }
gfCNCPoint2[9151] = {X 209.6277, Y 71.7691, Z -3.0000, A 0.000, B 0.000, C 0.000 }
gfCNCPoint2[9152] = {X 208.1881, Y 70.9077, Z -3.0000, A 0.000, B 0.000, C 0.000 }
gfCNCPoint2[9153] = {X 206.8579, Y 69.8855, Z -3.0000, A 0.000, B 0.000, C 0.000 }
gfCNCPoint2[9154] = {X 205.6547, Y 68.7163, Z -3.0000, A 0.000, B 0.000, C 0.000 }
gfCNCPoint2[9155] = {X 204.5949, Y 67.4158, Z -3.0000, A 0.000, B 0.000, C 0.000 }
gfCNCPoint2[9156] = {X 203.6927, Y 66.0015, Z -3.0000, A 0.000, B 0.000, C 0.000 }
gfCNCPoint2[9157] = {X 202.9600, Y 64.4923, Z -3.0000, A 0.000, B 0.000, C 0.000 }
gfCNCPoint2[9158] = {X 202.4069, Y 62.9084, Z -3.0000, A 0.000, B 0.000, C 0.000 }
gfCNCPoint2[9159] = {X 202.0407, Y 61.2713, Z -3.0000, A 0.000, B 0.000, C 0.000 }
gfCNCPoint2[9160] = {X 199.6721, Y 61.6586, Z -3.0000, A 0.000, B 0.000, C 0.000 }
gfCNCPoint2[9161] = {X 199.5095, Y 60.3405, Z -3.0000, A 0.000, B 0.000, C 0.000 }
gfCNCPoint2[9162] = {X 199.4510, Y 59.0136, Z -3.0000, A 0.000, B 0.000, C 0.000 }
gfCNCPoint2[9163] = {X 199.4508, Y 58.0000, Z -3.0000, A 0.000, B 0.000, C 0.000 }
gfCNCPoint2[9164] = {X 199.5412, Y 56.2554, Z -3.0000, A 0.000, B 0.000, C 0.000 }
gfCNCPoint2[9165] = {X 199.8114, Y 54.5296, Z -3.0000, A 0.000, B 0.000, C 0.000 }
gfCNCPoint2[9166] = {X 197.5977, Y 55.4808, Z -3.0000, A 0.000, B 0.000, C 0.000 }
gfCNCPoint2[9167] = {X 195.3260, Y 56.2836, Z -3.0000, A 0.000, B 0.000, C 0.000 }
gfCNCPoint2[9168] = {X 195.3578, Y 56.6300, Z -3.0000, A 0.000, B 0.000, C 0.000 }
gfCNCPoint2[9169] = {X 195.3825, Y 56.9770, Z -3.0000, A 0.000, B 0.000, C 0.000 }
gfCNCPoint2[9170] = {X 199.6721, Y 61.6586, Z -3.0000, A 0.000, B 0.000, C 0.000 }
gfCNCPoint2[9171] = {X 202.0407, Y 61.2713, Z -3.0000, A 0.000, B 0.000, C 0.000 }
gfCNCPoint2[9172] = {X 201.9014, Y 60.1430, Z -3.0000, A 0.000, B 0.000, C 0.000 }
gfCNCPoint2[9173] = {X 201.8510, Y 59.0073, Z -3.0000, A 0.000, B 0.000, C 0.000 }
gfCNCPoint2[9174] = {X 201.8508, Y 58.0000, Z -3.0000, A 0.000, B 0.000, C 0.000 }
gfCNCPoint2[9175] = {X 201.9283, Y 56.5035, Z -3.0000, A 0.000, B 0.000, C 0.000 }
gfCNCPoint2[9176] = {X 202.1601, Y 55.0230, Z -3.0000, A 0.000, B 0.000, C 0.000 }
gfCNCPoint2[9177] = {X 202.4970, Y 53.7228, Z -3.0000, A 0.000, B 0.000, C 0.000 }
gfCNCPoint2[9178] = {X 202.9528, Y 52.4593, Z -3.0000, A 0.000, B 0.000, C 0.000 }
gfCNCPoint2[9179] = {X 203.5238, Y 51.2435, Z -3.0000, A 0.000, B 0.000, C 0.000 }
gfCNCPoint2[9180] = {X 202.2639, Y 51.6551, Z -3.0000, A 0.000, B 0.000, C 0.000 }
gfCNCPoint2[9181] = {X 200.9596, Y 51.8909, Z -3.0000, A 0.000, B 0.000, C 0.000 }
gfCNCPoint2[9182] = {X 199.6354, Y 51.9467, Z -3.0000, A 0.000, B 0.000, C 0.000 }
gfCNCPoint2[9183] = {X 199.2149, Y 52.1547, Z -3.0000, A 0.000, B 0.000, C 0.000 }
gfCNCPoint2[9184] = {X 198.7916, Y 52.3570, Z -3.0000, A 0.000, B 0.000, C 0.000 }
gfCNCPoint2[9185] = {X 196.7764, Y 53.2248, Z -3.0000, A 0.000, B 0.000, C 0.000 }
gfCNCPoint2[9186] = {X 194.7096, Y 53.9610, Z -3.0000, A 0.000, B 0.000, C 0.000 }
gfCNCPoint2[9187] = {X 192.5996, Y 54.5626, Z -3.0000, A 0.000, B 0.000, C 0.000 }
gfCNCPoint2[9188] = {X 192.9063, Y 56.2411, Z -3.0000, A 0.000, B 0.000, C 0.000 }
gfCNCPoint2[9189] = {X 193.0134, Y 57.9440, Z -3.0000, A 0.000, B 0.000, C 0.000 }
gfCNCPoint2[9190] = {X 210.3943, Y 76.9130, Z -3.0000, A 0.000, B 0.000, C 0.000 }
gfCNCPoint2[9191] = {X 208.6248, Y 78.5344, Z -3.0000, A 0.000, B 0.000, C 0.000 }
gfCNCPoint2[9192] = {X 214.3884, Y 84.8247, Z -3.0000, A 0.000, B 0.000, C 0.000 }
gfCNCPoint2[9193] = {X 228.8378, Y 75.5677, Z -3.0000, A 0.000, B 0.000, C 0.000 }
gfCNCPoint2[9194] = {X 218.7731, Y 71.6178, Z -3.0000, A 0.000, B 0.000, C 0.000 }
gfCNCPoint2[9195] = {X 217.8434, Y 71.3041, Z -3.0000, A 0.000, B 0.000, C 0.000 }
gfCNCPoint2[9196] = {X 216.8839, Y 71.0995, Z -3.0000, A 0.000, B 0.000, C 0.000 }
gfCNCPoint2[9197] = {X 215.9071, Y 71.0066, Z -3.0000, A 0.000, B 0.000, C 0.000 }
gfCNCPoint2[9198] = {X 214.2372, Y 70.8313, Z -3.0000, A 0.000, B 0.000, C 0.000 }
gfCNCPoint2[9199] = {X 212.6078, Y 70.4260, Z -3.0000, A 0.000, B 0.000, C 0.000 }
gfCNCPoint2[9200] = {X 211.0502, Y 69.7988, Z -3.0000, A 0.000, B 0.000, C 0.000 }
gfCNCPoint2[9201] = {X 209.5947, Y 68.9616, Z -3.0000, A 0.000, B 0.000, C 0.000 }
gfCNCPoint2[9202] = {X 208.2693, Y 67.9307, Z -3.0000, A 0.000, B 0.000, C 0.000 }
gfCNCPoint2[9203] = {X 207.0997, Y 66.7260, Z -3.0000, A 0.000, B 0.000, C 0.000 }
gfCNCPoint2[9204] = {X 206.1084, Y 65.3707, Z -3.0000, A 0.000, B 0.000, C 0.000 }
gfCNCPoint2[9205] = {X 205.3147, Y 63.8910, Z -3.0000, A 0.000, B 0.000, C 0.000 }
gfCNCPoint2[9206] = {X 204.7338, Y 62.3156, Z -3.0000, A 0.000, B 0.000, C 0.000 }
gfCNCPoint2[9207] = {X 204.3769, Y 60.6749, Z -3.0000, A 0.000, B 0.000, C 0.000 }
gfCNCPoint2[9208] = {X 204.2510, Y 59.0005, Z -3.0000, A 0.000, B 0.000, C 0.000 }
gfCNCPoint2[9209] = {X 204.2508, Y 58.0000, Z -3.0000, A 0.000, B 0.000, C 0.000 }
gfCNCPoint2[9210] = {X 204.3397, Y 56.5375, Z -3.0000, A 0.000, B 0.000, C 0.000 }
gfCNCPoint2[9211] = {X 204.6049, Y 55.0966, Z -3.0000, A 0.000, B 0.000, C 0.000 }
gfCNCPoint2[9212] = {X 205.0427, Y 53.6984, Z -3.0000, A 0.000, B 0.000, C 0.000 }
gfCNCPoint2[9213] = {X 205.6465, Y 52.3634, Z -3.0000, A 0.000, B 0.000, C 0.000 }
gfCNCPoint2[9214] = {X 206.5300, Y 50.9381, Z -3.0000, A 0.000, B 0.000, C 0.000 }
gfCNCPoint2[9215] = {X 207.6023, Y 49.6490, Z -3.0000, A 0.000, B 0.000, C 0.000 }
gfCNCPoint2[9216] = {X 208.8428, Y 48.5207, Z -3.0000, A 0.000, B 0.000, C 0.000 }
gfCNCPoint2[9217] = {X 210.2277, Y 47.5751, Z -3.0000, A 0.000, B 0.000, C 0.000 }
gfCNCPoint2[9218] = {X 209.8801, Y 46.3328, Z -3.0000, A 0.000, B 0.000, C 0.000 }
gfCNCPoint2[9219] = {X 209.7572, Y 45.0487, Z -3.0000, A 0.000, B 0.000, C 0.000 }
gfCNCPoint2[9220] = {X 209.7570, Y 44.1980, Z -3.0000, A 0.000, B 0.000, C 0.000 }
gfCNCPoint2[9221] = {X 209.8559, Y 43.0076, Z -3.0000, A 0.000, B 0.000, C 0.000 }
gfCNCPoint2[9222] = {X 210.1498, Y 41.8499, Z -3.0000, A 0.000, B 0.000, C 0.000 }
gfCNCPoint2[9223] = {X 210.6308, Y 40.7565, Z -3.0000, A 0.000, B 0.000, C 0.000 }
gfCNCPoint2[9224] = {X 211.2855, Y 39.7574, Z -3.0000, A 0.000, B 0.000, C 0.000 }
gfCNCPoint2[9225] = {X 211.2855, Y 37.0782, Z -3.0000, A 0.000, B 0.000, C 0.000 }
gfCNCPoint2[9226] = {X 211.2853, Y 17.4407, Z -3.0000, A 0.000, B 0.000, C 0.000 }
gfCNCPoint2[9227] = {X 210.6366, Y 16.4468, Z -3.0000, A 0.000, B 0.000, C 0.000 }
gfCNCPoint2[9228] = {X 210.1580, Y 15.3607, Z -3.0000, A 0.000, B 0.000, C 0.000 }
gfCNCPoint2[9229] = {X 209.8622, Y 14.2113, Z -3.0000, A 0.000, B 0.000, C 0.000 }
gfCNCPoint2[9230] = {X 209.7572, Y 13.0291, Z -3.0000, A 0.000, B 0.000, C 0.000 }
gfCNCPoint2[9231] = {X 209.7570, Y 12.1868, Z -3.0000, A 0.000, B 0.000, C 0.000 }
gfCNCPoint2[9232] = {X 209.7578, Y 12.0808, Z -3.0000, A 0.000, B 0.000, C 0.000 }
gfCNCPoint2[9233] = {X 209.7601, Y 11.9749, Z -3.0000, A 0.000, B 0.000, C 0.000 }
gfCNCPoint2[9234] = {X 209.9068, Y 10.7178, Z -3.0000, A 0.000, B 0.000, C 0.000 }
gfCNCPoint2[9235] = {X 210.2690, Y 9.5050, Z -3.0000, A 0.000, B 0.000, C 0.000 }
gfCNCPoint2[9236] = {X 207.3611, Y 9.5050, Z -3.0000, A 0.000, B 0.000, C 0.000 }
gfCNCPoint2[9237] = {X 207.3611, Y 7.1050, Z -3.0000, A 0.000, B 0.000, C 0.000 }
gfCNCPoint2[9238] = {X 191.1439, Y 7.1050, Z -3.0000, A 0.000, B 0.000, C 0.000 }
gfCNCPoint2[9239] = {X 193.1008, Y 7.6484, Z -3.0000, A 0.000, B 0.000, C 0.000 }
gfCNCPoint2[9240] = {X 194.9840, Y 8.4085, Z -3.0000, A 0.000, B 0.000, C 0.000 }
gfCNCPoint2[9241] = {X 196.7697, Y 9.3759, Z -3.0000, A 0.000, B 0.000, C 0.000 }
gfCNCPoint2[9242] = {X 198.4352, Y 10.5381, Z -3.0000, A 0.000, B 0.000, C 0.000 }
gfCNCPoint2[9243] = {X 198.8572, Y 10.8885, Z -3.0000, A 0.000, B 0.000, C 0.000 }
gfCNCPoint2[9244] = {X 199.2647, Y 11.2556, Z -3.0000, A 0.000, B 0.000, C 0.000 }
gfCNCPoint2[9245] = {X 200.3497, Y 12.3982, Z -3.0000, A 0.000, B 0.000, C 0.000 }
gfCNCPoint2[9246] = {X 201.2953, Y 13.6586, Z -3.0000, A 0.000, B 0.000, C 0.000 }
gfCNCPoint2[9247] = {X 202.0889, Y 15.0198, Z -3.0000, A 0.000, B 0.000, C 0.000 }
gfCNCPoint2[9248] = {X 202.7198, Y 16.4636, Z -3.0000, A 0.000, B 0.000, C 0.000 }
gfCNCPoint2[9249] = {X 203.2136, Y 18.1834, Z -3.0000, A 0.000, B 0.000, C 0.000 }
gfCNCPoint2[9250] = {X 203.5069, Y 19.9484, Z -3.0000, A 0.000, B 0.000, C 0.000 }
gfCNCPoint2[9251] = {X 203.5960, Y 21.7354, Z -3.0000, A 0.000, B 0.000, C 0.000 }
gfCNCPoint2[9252] = {X 203.4797, Y 23.5208, Z -3.0000, A 0.000, B 0.000, C 0.000 }
gfCNCPoint2[9253] = {X 203.1594, Y 25.2812, Z -3.0000, A 0.000, B 0.000, C 0.000 }
gfCNCPoint2[9254] = {X 202.7591, Y 26.6265, Z -3.0000, A 0.000, B 0.000, C 0.000 }
gfCNCPoint2[9255] = {X 202.2075, Y 27.9172, Z -3.0000, A 0.000, B 0.000, C 0.000 }
gfCNCPoint2[9256] = {X 201.5119, Y 29.1364, Z -3.0000, A 0.000, B 0.000, C 0.000 }
gfCNCPoint2[9257] = {X 200.6815, Y 30.2680, Z -3.0000, A 0.000, B 0.000, C 0.000 }
gfCNCPoint2[9258] = {X 199.7270, Y 31.2972, Z -3.0000, A 0.000, B 0.000, C 0.000 }
gfCNCPoint2[9259] = {X 200.5666, Y 31.8697, Z -3.0000, A 0.000, B 0.000, C 0.000 }
gfCNCPoint2[9260] = {X 201.2695, Y 32.6037, Z -3.0000, A 0.000, B 0.000, C 0.000 }
gfCNCPoint2[9261] = {X 201.8050, Y 33.4673, Z -3.0000, A 0.000, B 0.000, C 0.000 }
gfCNCPoint2[9262] = {X 204.8262, Y 39.7091, Z -3.0000, A 0.000, B 0.000, C 0.000 }
gfCNCPoint2[9263] = {X 205.1508, Y 40.5847, Z -3.0000, A 0.000, B 0.000, C 0.000 }
gfCNCPoint2[9264] = {X 205.3026, Y 41.5062, Z -3.0000, A 0.000, B 0.000, C 0.000 }
gfCNCPoint2[9265] = {X 205.2761, Y 42.4397, Z -3.0000, A 0.000, B 0.000, C 0.000 }
gfCNCPoint2[9266] = {X 205.0723, Y 43.3511, Z -3.0000, A 0.000, B 0.000, C 0.000 }
gfCNCPoint2[9267] = {X 204.6986, Y 44.2070, Z -3.0000, A 0.000, B 0.000, C 0.000 }
gfCNCPoint2[9268] = {X 204.1687, Y 44.9760, Z -3.0000, A 0.000, B 0.000, C 0.000 }
gfCNCPoint2[9269] = {X 203.5020, Y 45.6299, Z -3.0000, A 0.000, B 0.000, C 0.000 }
gfCNCPoint2[9270] = {X 202.9656, Y 46.0636, Z -3.0000, A 0.000, B 0.000, C 0.000 }
gfCNCPoint2[9271] = {X 202.2135, Y 46.5638, Z -3.0000, A 0.000, B 0.000, C 0.000 }
gfCNCPoint2[9272] = {X 201.3822, Y 46.9172, Z -3.0000, A 0.000, B 0.000, C 0.000 }
gfCNCPoint2[9273] = {X 200.5002, Y 47.1119, Z -3.0000, A 0.000, B 0.000, C 0.000 }
gfCNCPoint2[9274] = {X 199.5974, Y 47.1412, Z -3.0000, A 0.000, B 0.000, C 0.000 }
gfCNCPoint2[9275] = {X 198.7046, Y 47.0042, Z -3.0000, A 0.000, B 0.000, C 0.000 }
gfCNCPoint2[9276] = {X 196.3904, Y 48.1787, Z -3.0000, A 0.000, B 0.000, C 0.000 }
gfCNCPoint2[9277] = {X 193.9811, Y 49.1435, Z -3.0000, A 0.000, B 0.000, C 0.000 }
gfCNCPoint2[9278] = {X 191.4959, Y 49.8910, Z -3.0000, A 0.000, B 0.000, C 0.000 }
gfCNCPoint2[9279] = {X 190.2925, Y 50.1566, Z -3.0000, A 0.000, B 0.000, C 0.000 }
gfCNCPoint2[9280] = {X 189.0767, Y 50.3580, Z -3.0000, A 0.000, B 0.000, C 0.000 }
gfCNCPoint2[9281] = {X 186.8982, Y 50.5556, Z -3.0000, A 0.000, B 0.000, C 0.000 }
gfCNCPoint2[9282] = {X 184.7107, Y 50.5472, Z -3.0000, A 0.000, B 0.000, C 0.000 }
gfCNCPoint2[9283] = {X 184.7352, Y 50.0678, Z -3.0000, A 0.000, B 0.000, C 0.000 }
gfCNCPoint2[9284] = {X 183.1151, Y 49.9269, Z -3.0000, A 0.000, B 0.000, C 0.000 }
gfCNCPoint2[9285] = {X 181.5093, Y 49.6706, Z -3.0000, A 0.000, B 0.000, C 0.000 }
gfCNCPoint2[9286] = {X 179.6141, Y 49.1968, Z -3.0000, A 0.000, B 0.000, C 0.000 }
gfCNCPoint2[9287] = {X 177.7853, Y 48.5102, Z -3.0000, A 0.000, B 0.000, C 0.000 }
gfCNCPoint2[9288] = {X 176.0466, Y 47.6196, Z -3.0000, A 0.000, B 0.000, C 0.000 }
gfCNCPoint2[9289] = {X 174.4207, Y 46.5368, Z -3.0000, A 0.000, B 0.000, C 0.000 }
gfCNCPoint2[9290] = {X 173.1807, Y 45.4901, Z -3.0000, A 0.000, B 0.000, C 0.000 }
gfCNCPoint2[9291] = {X 172.0772, Y 44.3004, Z -3.0000, A 0.000, B 0.000, C 0.000 }
gfCNCPoint2[9292] = {X 171.1266, Y 42.9852, Z -3.0000, A 0.000, B 0.000, C 0.000 }
gfCNCPoint2[9293] = {X 170.3430, Y 41.5642, Z -3.0000, A 0.000, B 0.000, C 0.000 }
gfCNCPoint2[9294] = {X 169.7381, Y 40.0585, Z -3.0000, A 0.000, B 0.000, C 0.000 }
gfCNCPoint2[9295] = {X 169.3209, Y 38.4903, Z -3.0000, A 0.000, B 0.000, C 0.000 }
gfCNCPoint2[9296] = {X 169.0976, Y 36.8830, Z -3.0000, A 0.000, B 0.000, C 0.000 }
gfCNCPoint2[9297] = {X 169.0132, Y 35.0395, Z -3.0000, A 0.000, B 0.000, C 0.000 }
gfCNCPoint2[9298] = {X 169.1602, Y 33.1998, Z -3.0000, A 0.000, B 0.000, C 0.000 }
gfCNCPoint2[9299] = {X 169.5363, Y 31.3930, Z -3.0000, A 0.000, B 0.000, C 0.000 }
gfCNCPoint2[9300] = {X 170.1356, Y 29.6475, Z -3.0000, A 0.000, B 0.000, C 0.000 }
gfCNCPoint2[9301] = {X 170.7628, Y 28.3598, Z -3.0000, A 0.000, B 0.000, C 0.000 }
gfCNCPoint2[9302] = {X 171.5527, Y 27.1651, Z -3.0000, A 0.000, B 0.000, C 0.000 }
gfCNCPoint2[9303] = {X 172.4920, Y 26.0838, Z -3.0000, A 0.000, B 0.000, C 0.000 }
gfCNCPoint2[9304] = {X 173.5644, Y 25.1344, Z -3.0000, A 0.000, B 0.000, C 0.000 }
gfCNCPoint2[9305] = {X 174.7516, Y 24.3332, Z -3.0000, A 0.000, B 0.000, C 0.000 }
gfCNCPoint2[9306] = {X 173.9914, Y 23.9229, Z -3.0000, A 0.000, B 0.000, C 0.000 }
gfCNCPoint2[9307] = {X 173.3260, Y 23.3720, Z -3.0000, A 0.000, B 0.000, C 0.000 }
gfCNCPoint2[9308] = {X 172.7810, Y 22.7017, Z -3.0000, A 0.000, B 0.000, C 0.000 }
gfCNCPoint2[9309] = {X 172.3776, Y 21.9378, Z -3.0000, A 0.000, B 0.000, C 0.000 }
gfCNCPoint2[9310] = {X 169.7664, Y 15.5423, Z -3.0000, A 0.000, B 0.000, C 0.000 }
gfCNCPoint2[9311] = {X 169.5126, Y 14.6752, Z -3.0000, A 0.000, B 0.000, C 0.000 }
gfCNCPoint2[9312] = {X 169.4412, Y 13.7745, Z -3.0000, A 0.000, B 0.000, C 0.000 }
gfCNCPoint2[9313] = {X 169.5553, Y 12.8782, Z -3.0000, A 0.000, B 0.000, C 0.000 }
gfCNCPoint2[9314] = {X 169.8501, Y 12.0242, Z -3.0000, A 0.000, B 0.000, C 0.000 }
gfCNCPoint2[9315] = {X 170.3131, Y 11.2483, Z -3.0000, A 0.000, B 0.000, C 0.000 }
gfCNCPoint2[9316] = {X 170.9248, Y 10.5834, Z -3.0000, A 0.000, B 0.000, C 0.000 }
gfCNCPoint2[9317] = {X 171.6594, Y 10.0574, Z -3.0000, A 0.000, B 0.000, C 0.000 }
gfCNCPoint2[9318] = {X 172.2916, Y 9.6970, Z -3.0000, A 0.000, B 0.000, C 0.000 }
gfCNCPoint2[9319] = {X 173.1812, Y 9.3215, Z -3.0000, A 0.000, B 0.000, C 0.000 }
gfCNCPoint2[9320] = {X 174.1312, Y 9.1491, Z -3.0000, A 0.000, B 0.000, C 0.000 }
gfCNCPoint2[9321] = {X 175.0960, Y 9.1881, Z -3.0000, A 0.000, B 0.000, C 0.000 }
gfCNCPoint2[9322] = {X 176.0290, Y 9.4366, Z -3.0000, A 0.000, B 0.000, C 0.000 }
gfCNCPoint2[9323] = {X 178.2250, Y 8.5161, Z -3.0000, A 0.000, B 0.000, C 0.000 }
gfCNCPoint2[9324] = {X 180.5019, Y 7.8192, Z -3.0000, A 0.000, B 0.000, C 0.000 }
gfCNCPoint2[9325] = {X 182.8369, Y 7.3531, Z -3.0000, A 0.000, B 0.000, C 0.000 }
gfCNCPoint2[9326] = {X 185.2068, Y 7.1222, Z -3.0000, A 0.000, B 0.000, C 0.000 }
gfCNCPoint2[9327] = {X 187.5879, Y 7.1290, Z -3.0000, A 0.000, B 0.000, C 0.000 }
gfCNCPoint2[9328] = {X 189.9565, Y 7.3733, Z -3.0000, A 0.000, B 0.000, C 0.000 }
gfCNCPoint2[9329] = {X 191.7223, Y 7.7366, Z -3.0000, A 0.000, B 0.000, C 0.000 }
gfCNCPoint2[9330] = {X 193.4415, Y 8.2793, Z -3.0000, A 0.000, B 0.000, C 0.000 }
gfCNCPoint2[9331] = {X 195.0959, Y 8.9957, Z -3.0000, A 0.000, B 0.000, C 0.000 }
gfCNCPoint2[9332] = {X 196.6680, Y 9.8782, Z -3.0000, A 0.000, B 0.000, C 0.000 }
gfCNCPoint2[9333] = {X 198.1411, Y 10.9175, Z -3.0000, A 0.000, B 0.000, C 0.000 }
gfCNCPoint2[9334] = {X 199.2073, Y 11.8672, Z -3.0000, A 0.000, B 0.000, C 0.000 }
gfCNCPoint2[9335] = {X 200.1641, Y 12.9271, Z -3.0000, A 0.000, B 0.000, C 0.000 }
gfCNCPoint2[9336] = {X 201.0002, Y 14.0847, Z -3.0000, A 0.000, B 0.000, C 0.000 }
gfCNCPoint2[9337] = {X 201.7056, Y 15.3261, Z -3.0000, A 0.000, B 0.000, C 0.000 }
gfCNCPoint2[9338] = {X 202.2721, Y 16.6369, Z -3.0000, A 0.000, B 0.000, C 0.000 }
gfCNCPoint2[9339] = {X 202.7482, Y 18.3014, Z -3.0000, A 0.000, B 0.000, C 0.000 }
gfCNCPoint2[9340] = {X 203.0308, Y 20.0095, Z -3.0000, A 0.000, B 0.000, C 0.000 }
gfCNCPoint2[9341] = {X 203.1160, Y 21.7387, Z -3.0000, A 0.000, B 0.000, C 0.000 }
gfCNCPoint2[9342] = {X 203.0028, Y 23.4662, Z -3.0000, A 0.000, B 0.000, C 0.000 }
gfCNCPoint2[9343] = {X 202.6926, Y 25.1695, Z -3.0000, A 0.000, B 0.000, C 0.000 }
gfCNCPoint2[9344] = {X 202.2580, Y 26.5985, Z -3.0000, A 0.000, B 0.000, C 0.000 }
gfCNCPoint2[9345] = {X 201.6459, Y 27.9610, Z -3.0000, A 0.000, B 0.000, C 0.000 }
gfCNCPoint2[9346] = {X 200.8662, Y 29.2349, Z -3.0000, A 0.000, B 0.000, C 0.000 }
gfCNCPoint2[9347] = {X 199.9314, Y 30.3999, Z -3.0000, A 0.000, B 0.000, C 0.000 }
gfCNCPoint2[9348] = {X 198.8567, Y 31.4372, Z -3.0000, A 0.000, B 0.000, C 0.000 }
gfCNCPoint2[9349] = {X 199.6399, Y 31.7989, Z -3.0000, A 0.000, B 0.000, C 0.000 }
gfCNCPoint2[9350] = {X 200.3376, Y 32.3065, Z -3.0000, A 0.000, B 0.000, C 0.000 }
gfCNCPoint2[9351] = {X 200.9228, Y 32.9405, Z -3.0000, A 0.000, B 0.000, C 0.000 }
gfCNCPoint2[9352] = {X 201.3730, Y 33.6764, Z -3.0000, A 0.000, B 0.000, C 0.000 }
gfCNCPoint2[9353] = {X 204.3942, Y 39.9182, Z -3.0000, A 0.000, B 0.000, C 0.000 }
gfCNCPoint2[9354] = {X 204.7207, Y 40.8441, Z -3.0000, A 0.000, B 0.000, C 0.000 }
gfCNCPoint2[9355] = {X 204.8337, Y 41.8194, Z -3.0000, A 0.000, B 0.000, C 0.000 }
gfCNCPoint2[9356] = {X 204.7276, Y 42.7955, Z -3.0000, A 0.000, B 0.000, C 0.000 }
gfCNCPoint2[9357] = {X 204.4078, Y 43.7238, Z -3.0000, A 0.000, B 0.000, C 0.000 }
gfCNCPoint2[9358] = {X 203.8900, Y 44.5580, Z -3.0000, A 0.000, B 0.000, C 0.000 }
gfCNCPoint2[9359] = {X 203.2002, Y 45.2567, Z -3.0000, A 0.000, B 0.000, C 0.000 }
gfCNCPoint2[9360] = {X 202.6638, Y 45.6904, Z -3.0000, A 0.000, B 0.000, C 0.000 }
gfCNCPoint2[9361] = {X 201.9522, Y 46.1591, Z -3.0000, A 0.000, B 0.000, C 0.000 }
gfCNCPoint2[9362] = {X 201.1639, Y 46.4824, Z -3.0000, A 0.000, B 0.000, C 0.000 }
gfCNCPoint2[9363] = {X 200.3281, Y 46.6483, Z -3.0000, A 0.000, B 0.000, C 0.000 }
gfCNCPoint2[9364] = {X 199.4760, Y 46.6505, Z -3.0000, A 0.000, B 0.000, C 0.000 }
gfCNCPoint2[9365] = {X 198.6394, Y 46.4890, Z -3.0000, A 0.000, B 0.000, C 0.000 }
gfCNCPoint2[9366] = {X 196.3110, Y 47.6873, Z -3.0000, A 0.000, B 0.000, C 0.000 }
gfCNCPoint2[9367] = {X 193.8834, Y 48.6691, Z -3.0000, A 0.000, B 0.000, C 0.000 }
gfCNCPoint2[9368] = {X 191.3765, Y 49.4260, Z -3.0000, A 0.000, B 0.000, C 0.000 }
gfCNCPoint2[9369] = {X 189.1873, Y 49.8574, Z -3.0000, A 0.000, B 0.000, C 0.000 }
gfCNCPoint2[9370] = {X 186.9664, Y 50.0720, Z -3.0000, A 0.000, B 0.000, C 0.000 }
gfCNCPoint2[9371] = {X 184.7352, Y 50.0678, Z -3.0000, A 0.000, B 0.000, C 0.000 }
gfCNCPoint2[9372] = {X 184.7107, Y 50.5472, Z -3.0000, A 0.000, B 0.000, C 0.000 }
gfCNCPoint2[9373] = {X 185.7071, Y 51.5006, Z -3.0000, A 0.000, B 0.000, C 0.000 }
gfCNCPoint2[9374] = {X 186.5579, Y 52.5860, Z -3.0000, A 0.000, B 0.000, C 0.000 }
gfCNCPoint2[9375] = {X 187.2458, Y 53.7813, Z -3.0000, A 0.000, B 0.000, C 0.000 }
gfCNCPoint2[9376] = {X 187.7793, Y 55.1335, Z -3.0000, A 0.000, B 0.000, C 0.000 }
gfCNCPoint2[9377] = {X 188.1043, Y 56.5504, Z -3.0000, A 0.000, B 0.000, C 0.000 }
gfCNCPoint2[9378] = {X 188.2135, Y 58.0000, Z -3.0000, A 0.000, B 0.000, C 0.000 }
gfCNCPoint2[9379] = {X 188.2132, Y 59.0140, Z -3.0000, A 0.000, B 0.000, C 0.000 }
gfCNCPoint2[9380] = {X 188.2026, Y 59.3929, Z -3.0000, A 0.000, B 0.000, C 0.000 }
gfCNCPoint2[9381] = {X 188.1772, Y 59.7711, Z -3.0000, A 0.000, B 0.000, C 0.000 }
gfCNCPoint2[9382] = {X 213.5228, Y 87.4325, Z -3.0000, A 0.000, B 0.000, C 0.000 }
gfCNCPoint2[9383] = {X 214.2178, Y 87.3800, Z -3.0000, A 0.000, B 0.000, C 0.000 }
gfCNCPoint2[9384] = {X 214.9136, Y 87.3385, Z -3.0000, A 0.000, B 0.000, C 0.000 }
gfCNCPoint2[9385] = {X 234.0924, Y 75.0516, Z -3.0000, A 0.000, B 0.000, C 0.000 }
gfCNCPoint2[9386] = {X 219.6588, Y 69.3872, Z -3.0000, A 0.000, B 0.000, C 0.000 }
gfCNCPoint2[9387] = {X 218.4697, Y 68.9873, Z -3.0000, A 0.000, B 0.000, C 0.000 }
gfCNCPoint2[9388] = {X 217.2425, Y 68.7264, Z -3.0000, A 0.000, B 0.000, C 0.000 }
gfCNCPoint2[9389] = {X 215.9935, Y 68.6082, Z -3.0000, A 0.000, B 0.000, C 0.000 }
gfCNCPoint2[9390] = {X 214.5232, Y 68.4438, Z -3.0000, A 0.000, B 0.000, C 0.000 }
gfCNCPoint2[9391] = {X 213.0951, Y 68.0573, Z -3.0000, A 0.000, B 0.000, C 0.000 }
gfCNCPoint2[9392] = {X 211.7426, Y 67.4576, Z -3.0000, A 0.000, B 0.000, C 0.000 }
gfCNCPoint2[9393] = {X 210.4973, Y 66.6589, Z -3.0000, A 0.000, B 0.000, C 0.000 }
gfCNCPoint2[9394] = {X 209.3883, Y 65.6797, Z -3.0000, A 0.000, B 0.000, C 0.000 }
gfCNCPoint2[9395] = {X 208.4414, Y 64.5430, Z -3.0000, A 0.000, B 0.000, C 0.000 }
gfCNCPoint2[9396] = {X 207.6788, Y 63.2752, Z -3.0000, A 0.000, B 0.000, C 0.000 }
gfCNCPoint2[9397] = {X 207.1183, Y 61.9060, Z -3.0000, A 0.000, B 0.000, C 0.000 }
gfCNCPoint2[9398] = {X 206.7730, Y 60.4674, Z -3.0000, A 0.000, B 0.000, C 0.000 }
gfCNCPoint2[9399] = {X 206.6510, Y 58.9930, Z -3.0000, A 0.000, B 0.000, C 0.000 }
gfCNCPoint2[9400] = {X 206.6508, Y 58.0000, Z -3.0000, A 0.000, B 0.000, C 0.000 }
gfCNCPoint2[9401] = {X 206.7577, Y 56.5655, Z -3.0000, A 0.000, B 0.000, C 0.000 }
gfCNCPoint2[9402] = {X 207.0760, Y 55.1628, Z -3.0000, A 0.000, B 0.000, C 0.000 }
gfCNCPoint2[9403] = {X 207.5986, Y 53.8226, Z -3.0000, A 0.000, B 0.000, C 0.000 }
gfCNCPoint2[9404] = {X 208.3140, Y 52.5747, Z -3.0000, A 0.000, B 0.000, C 0.000 }
gfCNCPoint2[9405] = {X 209.2065, Y 51.4466, Z -3.0000, A 0.000, B 0.000, C 0.000 }
gfCNCPoint2[9406] = {X 210.2563, Y 50.4632, Z -3.0000, A 0.000, B 0.000, C 0.000 }
gfCNCPoint2[9407] = {X 211.4402, Y 49.6463, Z -3.0000, A 0.000, B 0.000, C 0.000 }
gfCNCPoint2[9408] = {X 212.5893, Y 49.0723, Z -3.0000, A 0.000, B 0.000, C 0.000 }
gfCNCPoint2[9409] = {X 213.8042, Y 48.6556, Z -3.0000, A 0.000, B 0.000, C 0.000 }
gfCNCPoint2[9410] = {X 213.2578, Y 48.0874, Z -3.0000, A 0.000, B 0.000, C 0.000 }
gfCNCPoint2[9411] = {X 212.8100, Y 47.4386, Z -3.0000, A 0.000, B 0.000, C 0.000 }
gfCNCPoint2[9412] = {X 212.4725, Y 46.7262, Z -3.0000, A 0.000, B 0.000, C 0.000 }
gfCNCPoint2[9413] = {X 212.2401, Y 45.8965, Z -3.0000, A 0.000, B 0.000, C 0.000 }
gfCNCPoint2[9414] = {X 212.1572, Y 45.0389, Z -3.0000, A 0.000, B 0.000, C 0.000 }
gfCNCPoint2[9415] = {X 212.1570, Y 44.1980, Z -3.0000, A 0.000, B 0.000, C 0.000 }
gfCNCPoint2[9416] = {X 212.2384, Y 43.3166, Z -3.0000, A 0.000, B 0.000, C 0.000 }
gfCNCPoint2[9417] = {X 212.4797, Y 42.4650, Z -3.0000, A 0.000, B 0.000, C 0.000 }
gfCNCPoint2[9418] = {X 212.8729, Y 41.6720, Z -3.0000, A 0.000, B 0.000, C 0.000 }
gfCNCPoint2[9419] = {X 213.4046, Y 40.9643, Z -3.0000, A 0.000, B 0.000, C 0.000 }
gfCNCPoint2[9420] = {X 213.6828, Y 40.6575, Z -3.0000, A 0.000, B 0.000, C 0.000 }
gfCNCPoint2[9421] = {X 213.6855, Y 40.3041, Z -3.0000, A 0.000, B 0.000, C 0.000 }
gfCNCPoint2[9422] = {X 213.6855, Y 17.4645, Z -3.0000, A 0.000, B 0.000, C 0.000 }
gfCNCPoint2[9423] = {X 213.6802, Y 16.7697, Z -3.0000, A 0.000, B 0.000, C 0.000 }
gfCNCPoint2[9424] = {X 213.6799, Y 16.5198, Z -3.0000, A 0.000, B 0.000, C 0.000 }
gfCNCPoint2[9425] = {X 213.0405, Y 15.7785, Z -3.0000, A 0.000, B 0.000, C 0.000 }
gfCNCPoint2[9426] = {X 212.5620, Y 14.9244, Z -3.0000, A 0.000, B 0.000, C 0.000 }
gfCNCPoint2[9427] = {X 212.2635, Y 13.9920, Z -3.0000, A 0.000, B 0.000, C 0.000 }
gfCNCPoint2[9428] = {X 212.1572, Y 13.0188, Z -3.0000, A 0.000, B 0.000, C 0.000 }
gfCNCPoint2[9429] = {X 212.1570, Y 12.1868, Z -3.0000, A 0.000, B 0.000, C 0.000 }
gfCNCPoint2[9430] = {X 212.2436, Y 11.2717, Z -3.0000, A 0.000, B 0.000, C 0.000 }
gfCNCPoint2[9431] = {X 212.5002, Y 10.3891, Z -3.0000, A 0.000, B 0.000, C 0.000 }
gfCNCPoint2[9432] = {X 212.9449, Y 9.5281, Z -3.0000, A 0.000, B 0.000, C 0.000 }
gfCNCPoint2[9433] = {X 213.5510, Y 8.7718, Z -3.0000, A 0.000, B 0.000, C 0.000 }
gfCNCPoint2[9434] = {X 214.2946, Y 8.1503, Z -3.0000, A 0.000, B 0.000, C 0.000 }
gfCNCPoint2[9435] = {X 215.1463, Y 7.6880, Z -3.0000, A 0.000, B 0.000, C 0.000 }
gfCNCPoint2[9436] = {X 216.0727, Y 7.4030, Z -3.0000, A 0.000, B 0.000, C 0.000 }
gfCNCPoint2[9437] = {X 217.0370, Y 7.3068, Z -3.0000, A 0.000, B 0.000, C 0.000 }
gfCNCPoint2[9438] = {X 223.4805, Y 7.3068, Z -3.0000, A 0.000, B 0.000, C 0.000 }
gfCNCPoint2[9439] = {X 224.4448, Y 7.4030, Z -3.0000, A 0.000, B 0.000, C 0.000 }
gfCNCPoint2[9440] = {X 225.3712, Y 7.6880, Z -3.0000, A 0.000, B 0.000, C 0.000 }
gfCNCPoint2[9441] = {X 226.2229, Y 8.1503, Z -3.0000, A 0.000, B 0.000, C 0.000 }
gfCNCPoint2[9442] = {X 226.9665, Y 8.7718, Z -3.0000, A 0.000, B 0.000, C 0.000 }
gfCNCPoint2[9443] = {X 227.5726, Y 9.5281, Z -3.0000, A 0.000, B 0.000, C 0.000 }
gfCNCPoint2[9444] = {X 228.0173, Y 10.3891, Z -3.0000, A 0.000, B 0.000, C 0.000 }
gfCNCPoint2[9445] = {X 228.2739, Y 11.2717, Z -3.0000, A 0.000, B 0.000, C 0.000 }
gfCNCPoint2[9446] = {X 228.3605, Y 12.1868, Z -3.0000, A 0.000, B 0.000, C 0.000 }
gfCNCPoint2[9447] = {X 228.3603, Y 13.0237, Z -3.0000, A 0.000, B 0.000, C 0.000 }
gfCNCPoint2[9448] = {X 228.2528, Y 13.9973, Z -3.0000, A 0.000, B 0.000, C 0.000 }
gfCNCPoint2[9449] = {X 227.9532, Y 14.9298, Z -3.0000, A 0.000, B 0.000, C 0.000 }
gfCNCPoint2[9450] = {X 227.4733, Y 15.7836, Z -3.0000, A 0.000, B 0.000, C 0.000 }
gfCNCPoint2[9451] = {X 226.8326, Y 16.5245, Z -3.0000, A 0.000, B 0.000, C 0.000 }
gfCNCPoint2[9452] = {X 226.8335, Y 40.6632, Z -3.0000, A 0.000, B 0.000, C 0.000 }
gfCNCPoint2[9453] = {X 227.4740, Y 41.4041, Z -3.0000, A 0.000, B 0.000, C 0.000 }
gfCNCPoint2[9454] = {X 227.9536, Y 42.2579, Z -3.0000, A 0.000, B 0.000, C 0.000 }
gfCNCPoint2[9455] = {X 228.2530, Y 43.1904, Z -3.0000, A 0.000, B 0.000, C 0.000 }
gfCNCPoint2[9456] = {X 228.3603, Y 44.1638, Z -3.0000, A 0.000, B 0.000, C 0.000 }
gfCNCPoint2[9457] = {X 228.3605, Y 45.0000, Z -3.0000, A 0.000, B 0.000, C 0.000 }
gfCNCPoint2[9458] = {X 228.3507, Y 45.3090, Z -3.0000, A 0.000, B 0.000, C 0.000 }
gfCNCPoint2[9459] = {X 228.3214, Y 45.6167, Z -3.0000, A 0.000, B 0.000, C 0.000 }
gfCNCPoint2[9460] = {X 228.0910, Y 46.5992, Z -3.0000, A 0.000, B 0.000, C 0.000 }
gfCNCPoint2[9461] = {X 227.6635, Y 47.5134, Z -3.0000, A 0.000, B 0.000, C 0.000 }
gfCNCPoint2[9462] = {X 227.0571, Y 48.3200, Z -3.0000, A 0.000, B 0.000, C 0.000 }
gfCNCPoint2[9463] = {X 226.7053, Y 47.9934, Z -3.0000, A 0.000, B 0.000, C 0.000 }
gfCNCPoint2[9464] = {X 226.0261, Y 48.5889, Z -3.0000, A 0.000, B 0.000, C 0.000 }
gfCNCPoint2[9465] = {X 225.2396, Y 49.0331, Z -3.0000, A 0.000, B 0.000, C 0.000 }
gfCNCPoint2[9466] = {X 224.3790, Y 49.3073, Z -3.0000, A 0.000, B 0.000, C 0.000 }
gfCNCPoint2[9467] = {X 223.4805, Y 49.4000, Z -3.0000, A 0.000, B 0.000, C 0.000 }
gfCNCPoint2[9468] = {X 217.0370, Y 49.4000, Z -3.0000, A 0.000, B 0.000, C 0.000 }
gfCNCPoint2[9469] = {X 216.0579, Y 49.2897, Z -3.0000, A 0.000, B 0.000, C 0.000 }
gfCNCPoint2[9470] = {X 215.1279, Y 48.9643, Z -3.0000, A 0.000, B 0.000, C 0.000 }
gfCNCPoint2[9471] = {X 214.2936, Y 48.4400, Z -3.0000, A 0.000, B 0.000, C 0.000 }
gfCNCPoint2[9472] = {X 213.5969, Y 47.7433, Z -3.0000, A 0.000, B 0.000, C 0.000 }
gfCNCPoint2[9473] = {X 213.0727, Y 46.9091, Z -3.0000, A 0.000, B 0.000, C 0.000 }
gfCNCPoint2[9474] = {X 212.7473, Y 45.9791, Z -3.0000, A 0.000, B 0.000, C 0.000 }
gfCNCPoint2[9475] = {X 212.6370, Y 45.0000, Z -3.0000, A 0.000, B 0.000, C 0.000 }
gfCNCPoint2[9476] = {X 212.6370, Y 44.1980, Z -3.0000, A 0.000, B 0.000, C 0.000 }
gfCNCPoint2[9477] = {X 212.7103, Y 43.4045, Z -3.0000, A 0.000, B 0.000, C 0.000 }
gfCNCPoint2[9478] = {X 212.9276, Y 42.6378, Z -3.0000, A 0.000, B 0.000, C 0.000 }
gfCNCPoint2[9479] = {X 213.2815, Y 41.9238, Z -3.0000, A 0.000, B 0.000, C 0.000 }
gfCNCPoint2[9480] = {X 213.7602, Y 41.2867, Z -3.0000, A 0.000, B 0.000, C 0.000 }
gfCNCPoint2[9481] = {X 214.1614, Y 40.8442, Z -3.0000, A 0.000, B 0.000, C 0.000 }
gfCNCPoint2[9482] = {X 214.1655, Y 40.3060, Z -3.0000, A 0.000, B 0.000, C 0.000 }
gfCNCPoint2[9483] = {X 214.1655, Y 17.4626, Z -3.0000, A 0.000, B 0.000, C 0.000 }
gfCNCPoint2[9484] = {X 214.1602, Y 16.7692, Z -3.0000, A 0.000, B 0.000, C 0.000 }
gfCNCPoint2[9485] = {X 214.1597, Y 16.3068, Z -3.0000, A 0.000, B 0.000, C 0.000 }
gfCNCPoint2[9486] = {X 213.5170, Y 15.6180, Z -3.0000, A 0.000, B 0.000, C 0.000 }
gfCNCPoint2[9487] = {X 213.0357, Y 14.8082, Z -3.0000, A 0.000, B 0.000, C 0.000 }
gfCNCPoint2[9488] = {X 212.7378, Y 13.9146, Z -3.0000, A 0.000, B 0.000, C 0.000 }
gfCNCPoint2[9489] = {X 212.6370, Y 12.9779, Z -3.0000, A 0.000, B 0.000, C 0.000 }
gfCNCPoint2[9490] = {X 212.6370, Y 12.1868, Z -3.0000, A 0.000, B 0.000, C 0.000 }
gfCNCPoint2[9491] = {X 212.7473, Y 11.2077, Z -3.0000, A 0.000, B 0.000, C 0.000 }
gfCNCPoint2[9492] = {X 213.0728, Y 10.2777, Z -3.0000, A 0.000, B 0.000, C 0.000 }
gfCNCPoint2[9493] = {X 213.5970, Y 9.4435, Z -3.0000, A 0.000, B 0.000, C 0.000 }
gfCNCPoint2[9494] = {X 214.2937, Y 8.7468, Z -3.0000, A 0.000, B 0.000, C 0.000 }
gfCNCPoint2[9495] = {X 215.1279, Y 8.2226, Z -3.0000, A 0.000, B 0.000, C 0.000 }
gfCNCPoint2[9496] = {X 216.0579, Y 7.8971, Z -3.0000, A 0.000, B 0.000, C 0.000 }
gfCNCPoint2[9497] = {X 217.0370, Y 7.7868, Z -3.0000, A 0.000, B 0.000, C 0.000 }
gfCNCPoint2[9498] = {X 223.4805, Y 7.7868, Z -3.0000, A 0.000, B 0.000, C 0.000 }
gfCNCPoint2[9499] = {X 224.4596, Y 7.8971, Z -3.0000, A 0.000, B 0.000, C 0.000 }
gfCNCPoint2[9500] = {X 225.3896, Y 8.2226, Z -3.0000, A 0.000, B 0.000, C 0.000 }
gfCNCPoint2[9501] = {X 226.2238, Y 8.7468, Z -3.0000, A 0.000, B 0.000, C 0.000 }
gfCNCPoint2[9502] = {X 226.9205, Y 9.4435, Z -3.0000, A 0.000, B 0.000, C 0.000 }
gfCNCPoint2[9503] = {X 227.4447, Y 10.2777, Z -3.0000, A 0.000, B 0.000, C 0.000 }
gfCNCPoint2[9504] = {X 227.7702, Y 11.2077, Z -3.0000, A 0.000, B 0.000, C 0.000 }
gfCNCPoint2[9505] = {X 227.8805, Y 12.1868, Z -3.0000, A 0.000, B 0.000, C 0.000 }
gfCNCPoint2[9506] = {X 227.8802, Y 13.0233, Z -3.0000, A 0.000, B 0.000, C 0.000 }
gfCNCPoint2[9507] = {X 227.7719, Y 13.9494, Z -3.0000, A 0.000, B 0.000, C 0.000 }
gfCNCPoint2[9508] = {X 227.4708, Y 14.8320, Z -3.0000, A 0.000, B 0.000, C 0.000 }
gfCNCPoint2[9509] = {X 226.9906, Y 15.6312, Z -3.0000, A 0.000, B 0.000, C 0.000 }
gfCNCPoint2[9510] = {X 226.3526, Y 16.3113, Z -3.0000, A 0.000, B 0.000, C 0.000 }
gfCNCPoint2[9511] = {X 226.3535, Y 40.8763, Z -3.0000, A 0.000, B 0.000, C 0.000 }
gfCNCPoint2[9512] = {X 226.9979, Y 41.5654, Z -3.0000, A 0.000, B 0.000, C 0.000 }
gfCNCPoint2[9513] = {X 227.4806, Y 42.3760, Z -3.0000, A 0.000, B 0.000, C 0.000 }
gfCNCPoint2[9514] = {X 227.7794, Y 43.2709, Z -3.0000, A 0.000, B 0.000, C 0.000 }
gfCNCPoint2[9515] = {X 227.8805, Y 44.2089, Z -3.0000, A 0.000, B 0.000, C 0.000 }
gfCNCPoint2[9516] = {X 227.8805, Y 45.0000, Z -3.0000, A 0.000, B 0.000, C 0.000 }
gfCNCPoint2[9517] = {X 227.8037, Y 45.8182, Z -3.0000, A 0.000, B 0.000, C 0.000 }
gfCNCPoint2[9518] = {X 227.5762, Y 46.6079, Z -3.0000, A 0.000, B 0.000, C 0.000 }
gfCNCPoint2[9519] = {X 227.2057, Y 47.3415, Z -3.0000, A 0.000, B 0.000, C 0.000 }
gfCNCPoint2[9520] = {X 226.7053, Y 47.9934, Z -3.0000, A 0.000, B 0.000, C 0.000 }
gfCNCPoint2[9521] = {X 227.0571, Y 48.3200, Z -3.0000, A 0.000, B 0.000, C 0.000 }
gfCNCPoint2[9522] = {X 236.2309, Y 48.3200, Z -3.0000, A 0.000, B 0.000, C 0.000 }
gfCNCPoint2[9523] = {X 235.6245, Y 47.5134, Z -3.0000, A 0.000, B 0.000, C 0.000 }
gfCNCPoint2[9524] = {X 235.1970, Y 46.5992, Z -3.0000, A 0.000, B 0.000, C 0.000 }
gfCNCPoint2[9525] = {X 234.9666, Y 45.6167, Z -3.0000, A 0.000, B 0.000, C 0.000 }
gfCNCPoint2[9526] = {X 234.9373, Y 45.3090, Z -3.0000, A 0.000, B 0.000, C 0.000 }
gfCNCPoint2[9527] = {X 234.9275, Y 45.0000, Z -3.0000, A 0.000, B 0.000, C 0.000 }
gfCNCPoint2[9528] = {X 234.9275, Y 44.2089, Z -3.0000, A 0.000, B 0.000, C 0.000 }
gfCNCPoint2[9529] = {X 235.0194, Y 43.2661, Z -3.0000, A 0.000, B 0.000, C 0.000 }
gfCNCPoint2[9530] = {X 235.2917, Y 42.3588, Z -3.0000, A 0.000, B 0.000, C 0.000 }
gfCNCPoint2[9531] = {X 235.7342, Y 41.5212, Z -3.0000, A 0.000, B 0.000, C 0.000 }
gfCNCPoint2[9532] = {X 236.3302, Y 40.7849, Z -3.0000, A 0.000, B 0.000, C 0.000 }
gfCNCPoint2[9533] = {X 237.0572, Y 40.1776, Z -3.0000, A 0.000, B 0.000, C 0.000 }
gfCNCPoint2[9534] = {X 237.8878, Y 39.7222, Z -3.0000, A 0.000, B 0.000, C 0.000 }
gfCNCPoint2[9535] = {X 241.5466, Y 32.5606, Z -3.0000, A 0.000, B 0.000, C 0.000 }
gfCNCPoint2[9536] = {X 240.2122, Y 31.5580, Z -3.0000, A 0.000, B 0.000, C 0.000 }
gfCNCPoint2[9537] = {X 239.0315, Y 30.3782, Z -3.0000, A 0.000, B 0.000, C 0.000 }
gfCNCPoint2[9538] = {X 238.0279, Y 29.0445, Z -3.0000, A 0.000, B 0.000, C 0.000 }
gfCNCPoint2[9539] = {X 237.2211, Y 27.5833, Z -3.0000, A 0.000, B 0.000, C 0.000 }
gfCNCPoint2[9540] = {X 236.6272, Y 26.0234, Z -3.0000, A 0.000, B 0.000, C 0.000 }
gfCNCPoint2[9541] = {X 236.1921, Y 24.1498, Z -3.0000, A 0.000, B 0.000, C 0.000 }
gfCNCPoint2[9542] = {X 235.9702, Y 22.2392, Z -3.0000, A 0.000, B 0.000, C 0.000 }
gfCNCPoint2[9543] = {X 235.9643, Y 20.3157, Z -3.0000, A 0.000, B 0.000, C 0.000 }
gfCNCPoint2[9544] = {X 236.1746, Y 18.4038, Z -3.0000, A 0.000, B 0.000, C 0.000 }
gfCNCPoint2[9545] = {X 236.5983, Y 16.5275, Z -3.0000, A 0.000, B 0.000, C 0.000 }
gfCNCPoint2[9546] = {X 237.1175, Y 15.0570, Z -3.0000, A 0.000, B 0.000, C 0.000 }
gfCNCPoint2[9547] = {X 237.8172, Y 13.6632, Z -3.0000, A 0.000, B 0.000, C 0.000 }
gfCNCPoint2[9548] = {X 238.6862, Y 12.3682, Z -3.0000, A 0.000, B 0.000, C 0.000 }
gfCNCPoint2[9549] = {X 239.7108, Y 11.1924, Z -3.0000, A 0.000, B 0.000, C 0.000 }
gfCNCPoint2[9550] = {X 240.8750, Y 10.1543, Z -3.0000, A 0.000, B 0.000, C 0.000 }
gfCNCPoint2[9551] = {X 242.1603, Y 9.2705, Z -3.0000, A 0.000, B 0.000, C 0.000 }
gfCNCPoint2[9552] = {X 243.5463, Y 8.5550, Z -3.0000, A 0.000, B 0.000, C 0.000 }
gfCNCPoint2[9553] = {X 245.0111, Y 8.0190, Z -3.0000, A 0.000, B 0.000, C 0.000 }
gfCNCPoint2[9554] = {X 246.5316, Y 7.6711, Z -3.0000, A 0.000, B 0.000, C 0.000 }
gfCNCPoint2[9555] = {X 248.6761, Y 7.3937, Z -3.0000, A 0.000, B 0.000, C 0.000 }
gfCNCPoint2[9556] = {X 250.8369, Y 7.3112, Z -3.0000, A 0.000, B 0.000, C 0.000 }
gfCNCPoint2[9557] = {X 266.7608, Y 7.3112, Z -3.0000, A 0.000, B 0.000, C 0.000 }
gfCNCPoint2[9558] = {X 267.7190, Y 7.4127, Z -3.0000, A 0.000, B 0.000, C 0.000 }
gfCNCPoint2[9559] = {X 268.6386, Y 7.7003, Z -3.0000, A 0.000, B 0.000, C 0.000 }
gfCNCPoint2[9560] = {X 269.4839, Y 8.1630, Z -3.0000, A 0.000, B 0.000, C 0.000 }
gfCNCPoint2[9561] = {X 270.2218, Y 8.7826, Z -3.0000, A 0.000, B 0.000, C 0.000 }
gfCNCPoint2[9562] = {X 270.8237, Y 9.5351, Z -3.0000, A 0.000, B 0.000, C 0.000 }
gfCNCPoint2[9563] = {X 271.2661, Y 10.3911, Z -3.0000, A 0.000, B 0.000, C 0.000 }
gfCNCPoint2[9564] = {X 271.5232, Y 11.2720, Z -3.0000, A 0.000, B 0.000, C 0.000 }
gfCNCPoint2[9565] = {X 271.6110, Y 12.1854, Z -3.0000, A 0.000, B 0.000, C 0.000 }
gfCNCPoint2[9566] = {X 271.6108, Y 13.0237, Z -3.0000, A 0.000, B 0.000, C 0.000 }
gfCNCPoint2[9567] = {X 271.5128, Y 13.9524, Z -3.0000, A 0.000, B 0.000, C 0.000 }
gfCNCPoint2[9568] = {X 271.2396, Y 14.8453, Z -3.0000, A 0.000, B 0.000, C 0.000 }
gfCNCPoint2[9569] = {X 275.6743, Y 16.6820, Z -3.0000, A 0.000, B 0.000, C 0.000 }
gfCNCPoint2[9570] = {X 275.3124, Y 17.4571, Z -3.0000, A 0.000, B 0.000, C 0.000 }
gfCNCPoint2[9571] = {X 274.8834, Y 18.1973, Z -3.0000, A 0.000, B 0.000, C 0.000 }
gfCNCPoint2[9572] = {X 274.8833, Y 38.9893, Z -3.0000, A 0.000, B 0.000, C 0.000 }
gfCNCPoint2[9573] = {X 275.3139, Y 39.7326, Z -3.0000, A 0.000, B 0.000, C 0.000 }
gfCNCPoint2[9574] = {X 275.6770, Y 40.5111, Z -3.0000, A 0.000, B 0.000, C 0.000 }
gfCNCPoint2[9575] = {X 276.0381, Y 39.7364, Z -3.0000, A 0.000, B 0.000, C 0.000 }
gfCNCPoint2[9576] = {X 276.4659, Y 38.9964, Z -3.0000, A 0.000, B 0.000, C 0.000 }
gfCNCPoint2[9577] = {X 276.4655, Y 18.1977, Z -3.0000, A 0.000, B 0.000, C 0.000 }
gfCNCPoint2[9578] = {X 276.0364, Y 17.4574, Z -3.0000, A 0.000, B 0.000, C 0.000 }
gfCNCPoint2[9579] = {X 275.6743, Y 16.6820, Z -3.0000, A 0.000, B 0.000, C 0.000 }
gfCNCPoint2[9580] = {X 273.4570, Y 15.7637, Z -3.0000, A 0.000, B 0.000, C 0.000 }
gfCNCPoint2[9581] = {X 273.0263, Y 16.6343, Z -3.0000, A 0.000, B 0.000, C 0.000 }
gfCNCPoint2[9582] = {X 272.4834, Y 17.4399, Z -3.0000, A 0.000, B 0.000, C 0.000 }
gfCNCPoint2[9583] = {X 272.4833, Y 39.7467, Z -3.0000, A 0.000, B 0.000, C 0.000 }
gfCNCPoint2[9584] = {X 273.0275, Y 40.5546, Z -3.0000, A 0.000, B 0.000, C 0.000 }
gfCNCPoint2[9585] = {X 273.4590, Y 41.4279, Z -3.0000, A 0.000, B 0.000, C 0.000 }
gfCNCPoint2[9586] = {X 273.7590, Y 42.3098, Z -3.0000, A 0.000, B 0.000, C 0.000 }
gfCNCPoint2[9587] = {X 273.9439, Y 43.2227, Z -3.0000, A 0.000, B 0.000, C 0.000 }
gfCNCPoint2[9588] = {X 274.0108, Y 44.1519, Z -3.0000, A 0.000, B 0.000, C 0.000 }
gfCNCPoint2[9589] = {X 274.0110, Y 45.0000, Z -3.0000, A 0.000, B 0.000, C 0.000 }
gfCNCPoint2[9590] = {X 273.9884, Y 45.5734, Z -3.0000, A 0.000, B 0.000, C 0.000 }
gfCNCPoint2[9591] = {X 273.9207, Y 46.1433, Z -3.0000, A 0.000, B 0.000, C 0.000 }
gfCNCPoint2[9592] = {X 275.0713, Y 45.9760, Z -3.0000, A 0.000, B 0.000, C 0.000 }
gfCNCPoint2[9593] = {X 276.2327, Y 45.9200, Z -3.0000, A 0.000, B 0.000, C 0.000 }
gfCNCPoint2[9594] = {X 277.3960, Y 45.9200, Z -3.0000, A 0.000, B 0.000, C 0.000 }
gfCNCPoint2[9595] = {X 277.3539, Y 45.4857, Z -3.0000, A 0.000, B 0.000, C 0.000 }
gfCNCPoint2[9596] = {X 277.3378, Y 45.0497, Z -3.0000, A 0.000, B 0.000, C 0.000 }
gfCNCPoint2[9597] = {X 277.3377, Y 44.1974, Z -3.0000, A 0.000, B 0.000, C 0.000 }
gfCNCPoint2[9598] = {X 277.4032, Y 43.2530, Z -3.0000, A 0.000, B 0.000, C 0.000 }
gfCNCPoint2[9599] = {X 277.5899, Y 42.3250, Z -3.0000, A 0.000, B 0.000, C 0.000 }
gfCNCPoint2[9600] = {X 277.8946, Y 41.4287, Z -3.0000, A 0.000, B 0.000, C 0.000 }
gfCNCPoint2[9601] = {X 278.3246, Y 40.5578, Z -3.0000, A 0.000, B 0.000, C 0.000 }
gfCNCPoint2[9602] = {X 278.8659, Y 39.7514, Z -3.0000, A 0.000, B 0.000, C 0.000 }
gfCNCPoint2[9603] = {X 278.8655, Y 17.4402, Z -3.0000, A 0.000, B 0.000, C 0.000 }
gfCNCPoint2[9604] = {X 278.3225, Y 16.6345, Z -3.0000, A 0.000, B 0.000, C 0.000 }
gfCNCPoint2[9605] = {X 277.8917, Y 15.7637, Z -3.0000, A 0.000, B 0.000, C 0.000 }
gfCNCPoint2[9606] = {X 277.5902, Y 14.8788, Z -3.0000, A 0.000, B 0.000, C 0.000 }
gfCNCPoint2[9607] = {X 277.4046, Y 13.9627, Z -3.0000, A 0.000, B 0.000, C 0.000 }
gfCNCPoint2[9608] = {X 277.3379, Y 13.0303, Z -3.0000, A 0.000, B 0.000, C 0.000 }
gfCNCPoint2[9609] = {X 277.3377, Y 12.1868, Z -3.0000, A 0.000, B 0.000, C 0.000 }
gfCNCPoint2[9610] = {X 277.3952, Y 11.2737, Z -3.0000, A 0.000, B 0.000, C 0.000 }
gfCNCPoint2[9611] = {X 277.5667, Y 10.3751, Z -3.0000, A 0.000, B 0.000, C 0.000 }
gfCNCPoint2[9612] = {X 277.8496, Y 9.5050, Z -3.0000, A 0.000, B 0.000, C 0.000 }
gfCNCPoint2[9613] = {X 273.4965, Y 9.5050, Z -3.0000, A 0.000, B 0.000, C 0.000 }
gfCNCPoint2[9614] = {X 273.7798, Y 10.3732, Z -3.0000, A 0.000, B 0.000, C 0.000 }
gfCNCPoint2[9615] = {X 273.9522, Y 11.2700, Z -3.0000, A 0.000, B 0.000, C 0.000 }
gfCNCPoint2[9616] = {X 274.0110, Y 12.1813, Z -3.0000, A 0.000, B 0.000, C 0.000 }
gfCNCPoint2[9617] = {X 274.0107, Y 13.0462, Z -3.0000, A 0.000, B 0.000, C 0.000 }
gfCNCPoint2[9618] = {X 273.9427, Y 13.9732, Z -3.0000, A 0.000, B 0.000, C 0.000 }
gfCNCPoint2[9619] = {X 273.7571, Y 14.8839, Z -3.0000, A 0.000, B 0.000, C 0.000 }
gfCNCPoint2[9620] = {X 273.4570, Y 15.7637, Z -3.0000, A 0.000, B 0.000, C 0.000 }
gfCNCPoint2[9621] = {X 271.2396, Y 14.8453, Z -3.0000, A 0.000, B 0.000, C 0.000 }
gfCNCPoint2[9622] = {X 270.7502, Y 15.7458, Z -3.0000, A 0.000, B 0.000, C 0.000 }
gfCNCPoint2[9623] = {X 270.0834, Y 16.5243, Z -3.0000, A 0.000, B 0.000, C 0.000 }
gfCNCPoint2[9624] = {X 270.0832, Y 40.6624, Z -3.0000, A 0.000, B 0.000, C 0.000 }
gfCNCPoint2[9625] = {X 270.7240, Y 41.4033, Z -3.0000, A 0.000, B 0.000, C 0.000 }
gfCNCPoint2[9626] = {X 271.2038, Y 42.2572, Z -3.0000, A 0.000, B 0.000, C 0.000 }
gfCNCPoint2[9627] = {X 271.5034, Y 43.1897, Z -3.0000, A 0.000, B 0.000, C 0.000 }
gfCNCPoint2[9628] = {X 271.6108, Y 44.1633, Z -3.0000, A 0.000, B 0.000, C 0.000 }
gfCNCPoint2[9629] = {X 271.6110, Y 45.0000, Z -3.0000, A 0.000, B 0.000, C 0.000 }
gfCNCPoint2[9630] = {X 271.5959, Y 45.3844, Z -3.0000, A 0.000, B 0.000, C 0.000 }
gfCNCPoint2[9631] = {X 271.5505, Y 45.7664, Z -3.0000, A 0.000, B 0.000, C 0.000 }
gfCNCPoint2[9632] = {X 271.2989, Y 46.7171, Z -3.0000, A 0.000, B 0.000, C 0.000 }
gfCNCPoint2[9633] = {X 270.8619, Y 47.5981, Z -3.0000, A 0.000, B 0.000, C 0.000 }
gfCNCPoint2[9634] = {X 270.2571, Y 48.3736, Z -3.0000, A 0.000, B 0.000, C 0.000 }
gfCNCPoint2[9635] = {X 269.5090, Y 49.0121, Z -3.0000, A 0.000, B 0.000, C 0.000 }
gfCNCPoint2[9636] = {X 268.6482, Y 49.4876, Z -3.0000, A 0.000, B 0.000, C 0.000 }
gfCNCPoint2[9637] = {X 267.7095, Y 49.7809, Z -3.0000, A 0.000, B 0.000, C 0.000 }
gfCNCPoint2[9638] = {X 266.7310, Y 49.8800, Z -3.0000, A 0.000, B 0.000, C 0.000 }
gfCNCPoint2[9639] = {X 262.1384, Y 49.8800, Z -3.0000, A 0.000, B 0.000, C 0.000 }
gfCNCPoint2[9640] = {X 262.1384, Y 54.6800, Z -3.0000, A 0.000, B 0.000, C 0.000 }
gfCNCPoint2[9641] = {X 260.2795, Y 54.6800, Z -3.0000, A 0.000, B 0.000, C 0.000 }
gfCNCPoint2[9642] = {X 261.9952, Y 55.3608, Z -3.0000, A 0.000, B 0.000, C 0.000 }
gfCNCPoint2[9643] = {X 262.0628, Y 55.0195, Z -3.0000, A 0.000, B 0.000, C 0.000 }
gfCNCPoint2[9644] = {X 262.1384, Y 54.6800, Z -3.0000, A 0.000, B 0.000, C 0.000 }
gfCNCPoint2[9645] = {X 262.1384, Y 52.2800, Z -3.0000, A 0.000, B 0.000, C 0.000 }
gfCNCPoint2[9646] = {X 260.2876, Y 52.2800, Z -3.0000, A 0.000, B 0.000, C 0.000 }
gfCNCPoint2[9647] = {X 259.1930, Y 52.1972, Z -3.0000, A 0.000, B 0.000, C 0.000 }
gfCNCPoint2[9648] = {X 258.1233, Y 51.9509, Z -3.0000, A 0.000, B 0.000, C 0.000 }
gfCNCPoint2[9649] = {X 257.1029, Y 51.5465, Z -3.0000, A 0.000, B 0.000, C 0.000 }
gfCNCPoint2[9650] = {X 256.1548, Y 50.9932, Z -3.0000, A 0.000, B 0.000, C 0.000 }
gfCNCPoint2[9651] = {X 255.3007, Y 50.3037, Z -3.0000, A 0.000, B 0.000, C 0.000 }
gfCNCPoint2[9652] = {X 253.6567, Y 52.0522, Z -3.0000, A 0.000, B 0.000, C 0.000 }
gfCNCPoint2[9653] = {X 253.4968, Y 51.8984, Z -3.0000, A 0.000, B 0.000, C 0.000 }
gfCNCPoint2[9654] = {X 253.3406, Y 51.7410, Z -3.0000, A 0.000, B 0.000, C 0.000 }
gfCNCPoint2[9655] = {X 253.2749, Y 51.8080, Z -3.0000, A 0.000, B 0.000, C 0.000 }
gfCNCPoint2[9656] = {X 253.2086, Y 51.8744, Z -3.0000, A 0.000, B 0.000, C 0.000 }
gfCNCPoint2[9657] = {X 253.6567, Y 52.0522, Z -3.0000, A 0.000, B 0.000, C 0.000 }
gfCNCPoint2[9658] = {X 255.3007, Y 50.3037, Z -3.0000, A 0.000, B 0.000, C 0.000 }
gfCNCPoint2[9659] = {X 255.1805, Y 50.1881, Z -3.0000, A 0.000, B 0.000, C 0.000 }
